KUKA KRL program: MyProgram_068().src

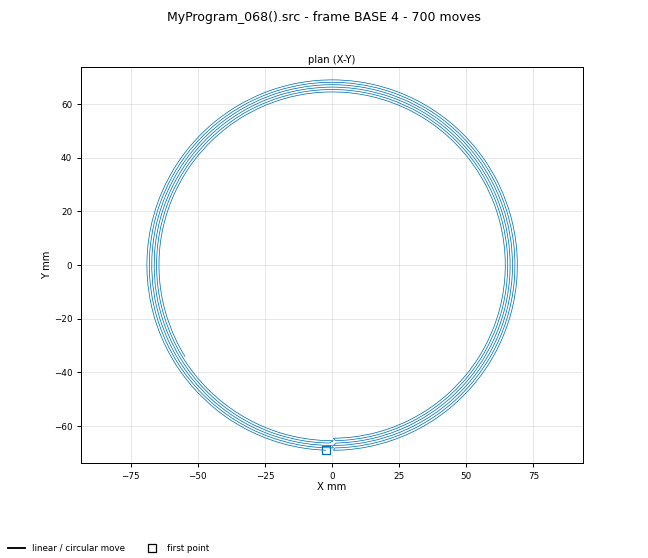
[picture p0: tool path of MyProgram_068().src in frame BASE 4, 700 of 700 moves have a stored position in this frame; points joined in program order, loops and branches not executed]
&ACCESS RVP
&REL 1
&PARAM TEMPLATE = C:\KRC\Roboter\Template\vorgabe
&PARAM EDITMASK = *
DEF MyProgram_068()
; ---- Setting reference (Base) ----
$BASE = BASE_DATA[4]

; --------------------------
; ---- Setting tool (TCP) ----
$TOOL = TOOL_DATA[3]
; --------------------------

$VEL.CP = VEL_APROX_PRINT
Startdeposition()
$VEL.CP = VEL_PRINT
LIN {X -2.4169,Y -68.9685,Z 75,A -97.7001,B 24.906,C -2.2384,E1 24.9936,E2 -177.965} C_DIS
LIN {X -6.7718,Y -68.6771,Z 75,A -101.3764,B 24.9061,C -2.2371,E1 24.9834,E2 -174.2842} C_DIS
LIN {X -9.1788,Y -68.3972,Z 75,A -103.4041,B 24.9061,C -2.2371,E1 24.9777,E2 -172.2549} C_DIS
LIN {X -12.2658,Y -67.9113,Z 75,A -106.3627,B 24.9068,C -2.2291,E1 24.9695,E2 -169.2747} C_DIS
LIN {X -15.7855,Y -67.181,Z 75,A -108.8346,B 24.9057,C -2.2426,E1 24.9629,E2 -166.8319} C_DIS
LIN {X -17.9152,Y -66.6442,Z 75,A -111.3209,B 24.9069,C -2.2281,E1 24.9561,E2 -164.3072} C_DIS
LIN {X -20.9966,Y -65.7389,Z 75,A -114.0064,B 24.9067,C -2.2296,E1 24.9489,E2 -161.6206} C_DIS
LIN {X -24.5799,Y -64.4845,Z 75,A -116.6949,B 24.9056,C -2.2431,E1 24.9419,E2 -158.9589} C_DIS
LIN {X -28.1955,Y -62.9876,Z 75,A -120.4389,B 24.9063,C -2.2351,E1 24.9322,E2 -155.187} C_DIS
LIN {X -31.9464,Y -61.1709,Z 75,A -123.1207,B 24.9044,C -2.2571,E1 24.9257,E2 -152.5506} C_DIS
LIN {X -33.7019,Y -60.2211,Z 75,A -125.4044,B 24.9055,C -2.245,E1 24.92,E2 -150.2315} C_DIS
LIN {X -37.4481,Y -57.9661,Z 75,A -128.5714,B 24.9041,C -2.2608,E1 24.9125,E2 -147.0923} C_DIS
LIN {X -39.6579,Y -56.4778,Z 75,A -131.4501,B 24.9051,C -2.2494,E1 24.9058,E2 -144.1767} C_DIS
LIN {X -42.7083,Y -54.2071,Z 75,A -134.5296,B 24.9045,C -2.2567,E1 24.899,E2 -141.1033} C_DIS
LIN {X -45.1659,Y -52.1779,Z 75,A -137.5073,B 24.9047,C -2.2544,E1 24.8927,E2 -138.1086} C_DIS
LIN {X -50.0115,Y -47.5541,Z 75,A -142.1725,B 24.902,C -2.2855,E1 24.8835,E2 -133.498} C_DIS
LIN {X -52.2098,Y -45.1287,Z 75,A -144.8753,B 24.9015,C -2.2919,E1 24.8785,E2 -130.7982} C_DIS
LIN {X -54.874,Y -41.8492,Z 75,A -148.4506,B 24.9009,C -2.2985,E1 24.8722,E2 -127.2221} C_DIS
LIN {X -56.1233,Y -40.157,Z 75,A -150.636,B 24.9013,C -2.2933,E1 24.8686,E2 -125.0136} C_DIS
LIN {X -57.9622,Y -37.4542,Z 75,A -153.0207,B 24.9001,C -2.3072,E1 24.8649,E2 -122.6502} C_DIS
LIN {X -59.1194,Y -35.6002,Z 75,A -156.0291,B 24.9019,C -2.2866,E1 24.8605,E2 -119.5771} C_DIS
LIN {X -61.0804,Y -32.1183,Z 75,A -159.2393,B 24.9009,C -2.2978,E1 24.8563,E2 -116.3766} C_DIS
LIN {X -62.7279,Y -28.7708,Z 75,A -161.5557,B 24.8988,C -2.3228,E1 24.8537,E2 -114.1072} C_DIS
LIN {X -64.116,Y -25.5271,Z 75,A -165.1655,B 24.8993,C -2.3169,E1 24.8498,E2 -110.4633} C_DIS
LIN {X -65.2783,Y -22.3892,Z 75,A -167.2138,B 24.8972,C -2.3402,E1 24.848,E2 -108.459} C_DIS
LIN {X -66.2797,Y -19.22,Z 75,A -169.9974,B 24.8966,C -2.3479,E1 24.8457,E2 -105.6777} C_DIS
LIN {X -67.1155,Y -16.059,Z 75,A -173.0277,B 24.8964,C -2.3495,E1 24.8436,E2 -102.6337} C_DIS
LIN {X -67.8136,Y -12.7977,Z 75,A -176.0352,B 24.8961,C -2.3531,E1 24.842,E2 -99.6169} C_DIS
LIN {X -68.5949,Y -7.5688,Z 75,A 178.9947,B 24.8959,C -2.3549,E1 24.8403,E2 -94.6213} C_DIS
LIN {X -68.9256,Y -3.4354,Z 75,A 176.9644,B 24.8924,C -2.3948,E1 24.84,E2 -92.6742} C_DIS
LIN {X -69.0119,Y -0.1041,Z 75,A 173.4964,B 24.8929,C -2.389,E1 24.8398,E2 -89.1714} C_DIS
LIN {X -68.9341,Y 3.2516,Z 75,A 170.7988,B 24.8919,C -2.3997,E1 24.8401,E2 -86.4831} C_DIS
LIN {X -68.597,Y 7.5488,Z 75,A 167.4395,B 24.8905,C -2.4155,E1 24.8409,E2 -83.1416} C_DIS
LIN {X -67.9375,Y 12.1205,Z 75,A 163.8781,B 24.8889,C -2.4334,E1 24.8424,E2 -79.6015} C_DIS
LIN {X -67.0696,Y 16.2506,Z 75,A 160.4913,B 24.8876,C -2.4468,E1 24.8444,E2 -76.2268} C_DIS
LIN {X -65.8431,Y 20.6675,Z 75,A 155.409,B 24.889,C -2.4322,E1 24.8484,E2 -71.0802} C_DIS
LIN {X -64.756,Y 23.8555,Z 75,A 153.2009,B 24.8871,C -2.4528,E1 24.8504,E2 -68.9088} C_DIS
LIN {X -63.907,Y 26.044,Z 75,A 150.9864,B 24.8871,C -2.4531,E1 24.8528,E2 -66.6829} C_DIS
LIN {X -62.007,Y 30.2934,Z 75,A 147.2256,B 24.8858,C -2.4667,E1 24.8572,E2 -62.934} C_DIS
LIN {X -59.24,Y 35.3996,Z 75,A 142.4927,B 24.8843,C -2.4823,E1 24.8636,E2 -58.2136} C_DIS
LIN {X -57.2828,Y 38.4856,Z 75,A 139.4955,B 24.8835,C -2.4915,E1 24.8682,E2 -55.2232} C_DIS
LIN {X -55.3718,Y 41.1877,Z 75,A 136.6952,B 24.8829,C -2.4977,E1 24.8728,E2 -52.4242} C_DIS
LIN {X -52.9777,Y 44.2243,Z 75,A 133.2143,B 24.8827,C -2.5003,E1 24.8789,E2 -48.9333} C_DIS
LIN {X -49.893,Y 47.6778,Z 75,A 130.0717,B 24.8803,C -2.5248,E1 24.8848,E2 -45.8351} C_DIS
LIN {X -47.8354,Y 49.7411,Z 75,A 126.9391,B 24.8812,C -2.5152,E1 24.8911,E2 -42.6666} C_DIS
LIN {X -45.1609,Y 52.1823,Z 75,A 123.1647,B 24.8822,C -2.5056,E1 24.8991,E2 -38.8544} C_DIS
LIN {X -41.8434,Y 54.8786,Z 75,A 119.5436,B 24.8816,C -2.5114,E1 24.9072,E2 -35.2341} C_DIS
LIN {X -38.259,Y 57.4348,Z 75,A 117.3549,B 24.8779,C -2.5502,E1 24.912,E2 -33.1306} C_DIS
LIN {X -35.8964,Y 58.9394,Z 75,A 114.595,B 24.8784,C -2.545,E1 24.9186,E2 -30.3494} C_DIS
LIN {X -32.8881,Y 60.6694,Z 75,A 111.7508,B 24.8779,C -2.5507,E1 24.9255,E2 -27.5107} C_DIS
LIN {X -27.9982,Y 63.0765,Z 75,A 106.5089,B 24.8787,C -2.5418,E1 24.9388,E2 -22.2343} C_DIS
LIN {X -24.9034,Y 64.3605,Z 75,A 104.6486,B 24.8764,C -2.5661,E1 24.9435,E2 -20.4278} C_DIS
LIN {X -22.9342,Y 65.0879,Z 75,A 102.0329,B 24.8781,C -2.5487,E1 24.9505,E2 -17.7655} C_DIS
LIN {X -19.8759,Y 66.0858,Z 75,A 99.9814,B 24.8764,C -2.5656,E1 24.9559,E2 -15.7507} C_DIS
LIN {X -15.4692,Y 67.254,Z 75,A 96.1652,B 24.8761,C -2.5685,E1 24.9662,E2 -11.9361} C_DIS
LIN {X -13.1799,Y 67.74,Z 75,A 93.4317,B 24.8777,C -2.552,E1 24.9739,E2 -9.1603} C_DIS
LIN {X -9.5408,Y 68.3476,Z 75,A 91.278,B 24.8755,C -2.5749,E1 24.9797,E2 -7.0592} C_DIS
LIN {X -6.6273,Y 68.6918,Z 75,A 88.761,B 24.8755,C -2.5743,E1 24.9866,E2 -4.5394} C_DIS
LIN {X -4.354,Y 68.8733,Z 75,A 85.9582,B 24.8776,C -2.5539,E1 24.9946,E2 -1.6871} C_DIS
LIN {X -0.5063,Y 69.0083,Z 75,A 83.6802,B 24.8754,C -2.5762,E1 25.0008,E2 0.5381} C_DIS
LIN {X 2.5422,Y 68.9643,Z 75,A 81.1062,B 24.8754,C -2.5754,E1 25.008,E2 3.1135} C_DIS
LIN {X 7.1724,Y 68.6364,Z 75,A 76.1587,B 24.878,C -2.5492,E1 25.0219,E2 8.1203} C_DIS
LIN {X 11.5572,Y 68.0357,Z 75,A 73.6683,B 24.8754,C -2.5764,E1 25.0286,E2 10.5438} C_DIS
LIN {X 14.4514,Y 67.4806,Z 75,A 70.6369,B 24.8769,C -2.5611,E1 25.037,E2 13.6075} C_DIS
LIN {X 17.8736,Y 66.6555,Z 75,A 67.8581,B 24.8767,C -2.5628,E1 25.0445,E2 16.378} C_DIS
LIN {X 21.6874,Y 65.5149,Z 75,A 65.1206,B 24.8756,C -2.5742,E1 25.0517,E2 19.0834} C_DIS
LIN {X 25.2023,Y 64.2436,Z 75,A 61.4768,B 24.8772,C -2.558,E1 25.0613,E2 22.758} C_DIS
LIN {X 29.4402,Y 62.4163,Z 75,A 58.0247,B 24.8767,C -2.5632,E1 25.07,E2 26.1892} C_DIS
LIN {X 32.7358,Y 60.752,Z 75,A 54.8729,B 24.8773,C -2.557,E1 25.0778,E2 29.3467} C_DIS
LIN {X 36.1577,Y 58.7806,Z 75,A 51.9971,B 24.8767,C -2.5626,E1 25.0847,E2 32.2007} C_DIS
LIN {X 39.1022,Y 56.864,Z 75,A 48.3317,B 24.879,C -2.5388,E1 25.0933,E2 35.9101} C_DIS
LIN {X 42.6741,Y 54.2341,Z 75,A 44.6835,B 24.8795,C -2.5332,E1 25.1014,E2 39.5582} C_DIS
LIN {X 45.0638,Y 52.2668,Z 75,A 42.5551,B 24.8789,C -2.5397,E1 25.1059,E2 41.6631} C_DIS
LIN {X 47.8326,Y 49.7438,Z 75,A 40.0156,B 24.8781,C -2.5484,E1 25.111,E2 44.1717} C_DIS
LIN {X 49.9659,Y 47.6021,Z 75,A 36.8259,B 24.8803,C -2.5252,E1 25.1173,E2 47.4026} C_DIS
LIN {X 53.072,Y 44.1108,Z 75,A 33.3588,B 24.8801,C -2.5273,E1 25.1237,E2 50.8491} C_DIS
LIN {X 55.6965,Y 40.7468,Z 75,A 28.9517,B 24.8831,C -2.496,E1 25.1312,E2 55.3092} C_DIS
LIN {X 57.6972,Y 37.861,Z 75,A 26.2056,B 24.8833,C -2.4931,E1 25.1354,E2 58.0486} C_DIS
LIN {X 60.3606,Y 33.4522,Z 75,A 22.0953,B 24.884,C -2.4862,E1 25.1411,E2 62.154} C_DIS
LIN {X 61.8517,Y 30.6067,Z 75,A 19.7892,B 24.8838,C -2.4886,E1 25.144,E2 64.4421} C_DIS
LIN {X 63.6158,Y 26.7475,Z 75,A 15.7389,B 24.886,C -2.4645,E1 25.1486,E2 68.5272} C_DIS
LIN {X 65.6592,Y 21.2431,Z 75,A 11.2518,B 24.8864,C -2.4607,E1 25.1527,E2 72.9981} C_DIS
LIN {X 66.648,Y 17.9012,Z 75,A 8.3955,B 24.8871,C -2.4531,E1 25.1549,E2 75.8561} C_DIS
LIN {X 67.5009,Y 14.3579,Z 75,A 5.5509,B 24.8875,C -2.4488,E1 25.1567,E2 78.6943} C_DIS
LIN {X 68.1413,Y 10.9181,Z 75,A 2.6382,B 24.8883,C -2.4396,E1 25.1581,E2 81.6117} C_DIS
LIN {X 68.6615,Y 6.9308,Z 75,A -0.3525,B 24.8883,C -2.4387,E1 25.1591,E2 84.5868} C_DIS
LIN {X 68.8098,Y 5.2596,Z 75,A -2.8449,B 24.8915,C -2.4044,E1 25.1596,E2 87.1454} C_DIS
LIN {X 68.9925,Y 1.593,Z 75,A -4.6966,B 24.8894,C -2.4273,E1 25.1598,E2 88.932} C_DIS
LIN {X 68.9365,Y -3.1965,Z 75,A -8.6973,B 24.8906,C -2.414,E1 25.1596,E2 92.9404} C_DIS
LIN {X 68.7647,Y -5.8221,Z 75,A -11.1863,B 24.892,C -2.3987,E1 25.1591,E2 95.4508} C_DIS
LIN {X 68.4631,Y -8.6741,Z 75,A -13.9477,B 24.8936,C -2.3808,E1 25.1581,E2 98.2382} C_DIS
LIN {X 67.7432,Y -13.1634,Z 75,A -17.5482,B 24.8943,C -2.3736,E1 25.1564,E2 101.8345} C_DIS
LIN {X 66.9693,Y -16.6615,Z 75,A -21.103,B 24.8965,C -2.3485,E1 25.154,E2 105.4279} C_DIS
LIN {X 65.9661,Y -20.2695,Z 75,A -23.5037,B 24.8957,C -2.3581,E1 25.1521,E2 107.7924} C_DIS
LIN {X 64.4258,Y -24.734,Z 75,A -27.5665,B 24.8971,C -2.3423,E1 25.1482,E2 111.8698} C_DIS
LIN {X 63.1759,Y -27.7714,Z 75,A -29.6765,B 24.8963,C -2.3509,E1 25.1459,E2 113.9479} C_DIS
LIN {X 61.2105,Y -31.8713,Z 75,A -34.8597,B 24.9006,C -2.3018,E1 25.1393,E2 119.2194} C_DIS
LIN {X 58.9736,Y -35.8402,Z 75,A -37.1636,B 24.8981,C -2.3308,E1 25.1362,E2 121.443} C_DIS
LIN {X 57.6967,Y -37.8618,Z 75,A -39.7177,B 24.8999,C -2.3099,E1 25.1322,E2 124.0336} C_DIS
LIN {X 55.38,Y -41.1773,Z 75,A -43.2595,B 24.9011,C -2.2959,E1 25.1264,E2 127.5914} C_DIS
LIN {X 52.7711,Y -44.4719,Z 75,A -46.2238,B 24.9007,C -2.3009,E1 25.1212,E2 130.5303} C_DIS
LIN {X 50.6612,Y -46.8606,Z 75,A -49.3423,B 24.9023,C -2.2817,E1 25.1153,E2 133.6804} C_DIS
LIN {X 46.7275,Y -50.7833,Z 75,A -53.2212,B 24.9016,C -2.2903,E1 25.1076,E2 137.5227} C_DIS
LIN {X 44.812,Y -52.4813,Z 75,A -55.5297,B 24.9024,C -2.2806,E1 25.1027,E2 139.845} C_DIS
LIN {X 42.6119,Y -54.2833,Z 75,A -58.3498,B 24.9039,C -2.2634,E1 25.0964,E2 142.6952} C_DIS
LIN {X 39.0721,Y -56.884,Z 75,A -61.6881,B 24.9039,C -2.2642,E1 25.0889,E2 146.0202} C_DIS
LIN {X 36.8921,Y -58.3226,Z 75,A -63.7241,B 24.9039,C -2.2635,E1 25.0841,E2 148.0512} C_DIS
LIN {X 34.1032,Y -59.9956,Z 75,A -67.0204,B 24.9056,C -2.2432,E1 25.076,E2 151.3856} C_DIS
LIN {X 30.9176,Y -61.6976,Z 75,A -70.0425,B 24.9061,C -2.2377,E1 25.0685,E2 154.4125} C_DIS
LIN {X 27.9422,Y -63.1014,Z 75,A -72.1201,B 24.905,C -2.2503,E1 25.0633,E2 156.4551} C_DIS
LIN {X 24.0168,Y -64.6973,Z 75,A -76.0525,B 24.9063,C -2.2349,E1 25.053,E2 160.4153} C_DIS
LIN {X 20.2897,Y -65.9602,Z 75,A -79.1443,B 24.9063,C -2.2355,E1 25.0448,E2 163.4999} C_DIS
LIN {X 15.7939,Y -67.179,Z 75,A -82.7107,B 24.9059,C -2.2392,E1 25.0352,E2 167.0521} C_DIS
LIN {X 11.2615,Y -68.0852,Z 75,A -86.5874,B 24.9063,C -2.2351,E1 25.0245,E2 170.9341} C_DIS
LIN {X 6.7327,Y -68.682,Z 75,A -90.3445,B 24.9064,C -2.2337,E1 25.0141,E2 174.6918} C_DIS
LIN {X 3.7919,Y -68.9059,Z 75,A -92.7846,B 24.9064,C -2.2328,E1 25.0073,E2 177.1329} C_DIS
LIN {X 0.4755,Y -68.972,Z 75,A -95.369,B 24.9061,C -2.2368,E1 25.0001,E2 179.7074} C_DIS
Enddeposition()
LIN {X 0.4755,Y -68.972,Z 75,A -95.369,B 24.9061,C -2.2368,E1 25.0001,E2 179.7074} C_DIS
Startdeposition()
$VEL.CP = VEL_PRINT
LIN {X 1.0869,Y -68.1022,Z 75,A -94.0872,B 24.9033,C -2.2708,E1 25.0039,E2 178.3451} C_DIS
LIN {X 3.4577,Y -68.0236,Z 75,A -91.8539,B 24.9027,C -2.2774,E1 25.0102,E2 176.0968} C_DIS
LIN {X 6.6528,Y -67.7862,Z 75,A -88.3869,B 24.9009,C -2.2981,E1 25.02,E2 172.5825} C_DIS
LIN {X 10.0513,Y -67.3654,Z 75,A -86.5018,B 24.9029,C -2.275,E1 25.025,E2 170.7541} C_DIS
LIN {X 14.6106,Y -66.5253,Z 75,A -82.5987,B 24.9026,C -2.2782,E1 25.0357,E2 166.8478} C_DIS
LIN {X 18.2097,Y -65.6324,Z 75,A -78.8592,B 24.901,C -2.2972,E1 25.0459,E2 163.069} C_DIS
LIN {X 21.6851,Y -64.5665,Z 75,A -75.0694,B 24.899,C -2.32,E1 25.0561,E2 159.2326} C_DIS
LIN {X 25.838,Y -63.0198,Z 75,A -72.1076,B 24.9003,C -2.3051,E1 25.0637,E2 156.3128} C_DIS
LIN {X 29.4896,Y -61.3957,Z 75,A -69.1878,B 24.9009,C -2.2988,E1 25.071,E2 153.4155} C_DIS
LIN {X 31.9355,Y -60.1602,Z 75,A -66.8974,B 24.9006,C -2.3022,E1 25.0767,E2 151.1232} C_DIS
LIN {X 34.9587,Y -58.4558,Z 75,A -63.9982,B 24.9002,C -2.3069,E1 25.0837,E2 148.2217} C_DIS
LIN {X 38.1825,Y -56.4018,Z 75,A -60.5693,B 24.8991,C -2.3187,E1 25.0917,E2 144.7761} C_DIS
LIN {X 41.0965,Y -54.3157,Z 75,A -57.5071,B 24.8985,C -2.3262,E1 25.0986,E2 141.7072} C_DIS
LIN {X 43.9939,Y -51.9967,Z 75,A -54.6941,B 24.8985,C -2.3248,E1 25.1047,E2 138.9082} C_DIS
LIN {X 45.5482,Y -50.6405,Z 75,A -52.7532,B 24.8978,C -2.3342,E1 25.1087,E2 136.9526} C_DIS
LIN {X 48.0466,Y -48.2769,Z 75,A -50.0508,B 24.8976,C -2.336,E1 25.1141,E2 134.2574} C_DIS
LIN {X 50.5842,Y -45.611,Z 75,A -47.0184,B 24.8971,C -2.3419,E1 25.1199,E2 131.2242} C_DIS
LIN {X 52.5069,Y -43.3836,Z 75,A -44.2671,B 24.8959,C -2.3558,E1 25.1249,E2 128.4529} C_DIS
LIN {X 54.7777,Y -40.4791,Z 75,A -41.181,B 24.8952,C -2.3636,E1 25.1301,E2 125.3629} C_DIS
LIN {X 57.5942,Y -36.3604,Z 75,A -37.5141,B 24.8954,C -2.3607,E1 25.1358,E2 121.721} C_DIS
LIN {X 59.0494,Y -33.9447,Z 75,A -34.8729,B 24.8942,C -2.3748,E1 25.1395,E2 119.0601} C_DIS
LIN {X 60.4973,Y -31.2932,Z 75,A -32.3896,B 24.8937,C -2.3806,E1 25.1428,E2 116.5762} C_DIS
LIN {X 61.731,Y -28.7812,Z 75,A -30.1209,B 24.8932,C -2.3852,E1 25.1455,E2 114.3087} C_DIS
LIN {X 62.7941,Y -26.3812,Z 75,A -27.627,B 24.8919,C -2.3997,E1 25.1483,E2 111.7944} C_DIS
LIN {X 64.3255,Y -22.3903,Z 75,A -24.4101,B 24.8919,C -2.4002,E1 25.1514,E2 108.5941} C_DIS
LIN {X 65.4179,Y -18.9657,Z 75,A -20.7689,B 24.8895,C -2.4266,E1 25.1544,E2 104.9113} C_DIS
LIN {X 66.4072,Y -15.1392,Z 75,A -17.7154,B 24.8892,C -2.4295,E1 25.1563,E2 101.8687} C_DIS
LIN {X 67.1595,Y -11.3437,Z 75,A -14.749,B 24.889,C -2.4318,E1 25.1578,E2 98.9142} C_DIS
LIN {X 67.6452,Y -7.9495,Z 75,A -12.1774,B 24.889,C -2.4324,E1 25.1588,E2 96.3564} C_DIS
LIN {X 67.8379,Y -6.0923,Z 75,A -10.3259,B 24.8878,C -2.4451,E1 25.1593,E2 94.4859} C_DIS
LIN {X 68.0448,Y -2.9954,Z 75,A -7.9509,B 24.8876,C -2.4469,E1 25.1597,E2 92.1207} C_DIS
LIN {X 68.0927,Y 1.6027,Z 75,A -4.3439,B 24.8872,C -2.4519,E1 25.1597,E2 88.5232} C_DIS
LIN {X 67.8357,Y 6.1162,Z 75,A 0.0289,B 24.8846,C -2.4795,E1 25.1589,E2 84.1113} C_DIS
LIN {X 67.5084,Y 9.0431,Z 75,A 2.642,B 24.8835,C -2.491,E1 25.158,E2 81.4865} C_DIS
LIN {X 66.6843,Y 13.8673,Z 75,A 6.4399,B 24.8832,C -2.4949,E1 25.1561,E2 77.7017} C_DIS
LIN {X 65.3548,Y 19.1795,Z 75,A 10.8866,B 24.8823,C -2.5043,E1 25.153,E2 73.2581} C_DIS
LIN {X 63.9617,Y 23.4088,Z 75,A 14.751,B 24.8809,C -2.5185,E1 25.1495,E2 69.382} C_DIS
LIN {X 62.5623,Y 26.9281,Z 75,A 18.2459,B 24.8793,C -2.536,E1 25.1457,E2 65.8651} C_DIS
LIN {X 60.827,Y 30.648,Z 75,A 21.9802,B 24.8776,C -2.5531,E1 25.1411,E2 62.1103} C_DIS
LIN {X 58.6332,Y 34.6586,Z 75,A 25.2658,B 24.8781,C -2.5482,E1 25.1366,E2 58.8533} C_DIS
LIN {X 56.754,Y 37.6576,Z 75,A 27.8055,B 24.8785,C -2.5441,E1 25.1328,E2 56.3361} C_DIS
LIN {X 54.7612,Y 40.5017,Z 75,A 31.5931,B 24.8756,C -2.5744,E1 25.1265,E2 52.4952} C_DIS
LIN {X 52.4107,Y 43.4993,Z 75,A 34.9365,B 24.8745,C -2.5855,E1 25.1206,E2 49.1409} C_DIS
LIN {X 50.2652,Y 45.9618,Z 75,A 36.5896,B 24.8767,C -2.5626,E1 25.1176,E2 47.5493} C_DIS
LIN {X 47.4872,Y 48.8275,Z 75,A 39.9639,B 24.876,C -2.5701,E1 25.111,E2 44.1717} C_DIS
LIN {X 44.8543,Y 51.2559,Z 75,A 42.7745,B 24.876,C -2.5709,E1 25.1053,E2 41.3706} C_DIS
LIN {X 42,Y 53.6205,Z 75,A 46.0803,B 24.8749,C -2.5815,E1 25.0981,E2 38.0523} C_DIS
LIN {X 39.2161,Y 55.6896,Z 75,A 50.0343,B 24.8718,C -2.6132,E1 25.089,E2 34.0371} C_DIS
LIN {X 36.5015,Y 57.505,Z 75,A 52.0993,B 24.8731,C -2.5999,E1 25.0843,E2 32.0104} C_DIS
LIN {X 34.0059,Y 59.0141,Z 75,A 54.7274,B 24.8723,C -2.6078,E1 25.0779,E2 29.3714} C_DIS
LIN {X 29.7678,Y 61.262,Z 75,A 58.4606,B 24.8726,C -2.6053,E1 25.0687,E2 25.6546} C_DIS
LIN {X 27.3322,Y 62.3862,Z 75,A 60.9801,B 24.8717,C -2.6144,E1 25.0622,E2 23.1197} C_DIS
LIN {X 23.6527,Y 63.8718,Z 75,A 64.3404,B 24.8713,C -2.6182,E1 25.0534,E2 19.7579} C_DIS
LIN {X 20.4574,Y 64.9666,Z 75,A 67.5673,B 24.8701,C -2.63,E1 25.0448,E2 16.5088} C_DIS
LIN {X 17.1421,Y 65.9186,Z 75,A 70.4294,B 24.8701,C -2.6308,E1 25.0371,E2 13.6493} C_DIS
LIN {X 12.4844,Y 66.958,Z 75,A 74.3353,B 24.8701,C -2.6298,E1 25.0264,E2 9.7504} C_DIS
LIN {X 6.9767,Y 67.7526,Z 75,A 78.7301,B 24.8707,C -2.6238,E1 25.0143,E2 5.3735} C_DIS
LIN {X 3.13,Y 68.0391,Z 75,A 81.7715,B 24.8712,C -2.6189,E1 25.0058,E2 2.3449} C_DIS
LIN {X -0.0016,Y 68.1119,Z 75,A 85.1275,B 24.8696,C -2.6357,E1 24.9964,E2 -1.0508} C_DIS
LIN {X -4.7805,Y 67.943,Z 75,A 88.9222,B 24.8702,C -2.6287,E1 24.9858,E2 -4.83} C_DIS
LIN {X -9.1383,Y 67.496,Z 75,A 93.0135,B 24.8695,C -2.6362,E1 24.9744,E2 -8.9419} C_DIS
LIN {X -12.7415,Y 66.9085,Z 75,A 95.0491,B 24.8721,C -2.6096,E1 24.969,E2 -10.9165} C_DIS
LIN {X -17.915,Y 65.7126,Z 75,A 99.6489,B 24.8722,C -2.6085,E1 24.9565,E2 -15.5199} C_DIS
LIN {X -21.2781,Y 64.7025,Z 75,A 102.4982,B 24.8728,C -2.6028,E1 24.949,E2 -18.3605} C_DIS
LIN {X -25.0973,Y 63.3185,Z 75,A 106.4735,B 24.872,C -2.611,E1 24.9385,E2 -22.3637} C_DIS
LIN {X -29.5209,Y 61.3807,Z 75,A 110.5312,B 24.8726,C -2.6048,E1 24.9282,E2 -26.4167} C_DIS
LIN {X -32.2641,Y 59.9846,Z 75,A 112.7631,B 24.8738,C -2.5925,E1 24.9228,E2 -28.6255} C_DIS
LIN {X -36.9014,Y 57.2484,Z 75,A 116.8402,B 24.8756,C -2.5744,E1 24.9131,E2 -32.6718} C_DIS
LIN {X -38.4899,Y 56.1932,Z 75,A 119.028,B 24.8746,C -2.5841,E1 24.9079,E2 -34.89} C_DIS
LIN {X -41.1422,Y 54.2815,Z 75,A 121.9427,B 24.8748,C -2.582,E1 24.9014,E2 -37.8103} C_DIS
LIN {X -44.6967,Y 51.3936,Z 75,A 125.4343,B 24.8764,C -2.5658,E1 24.894,E2 -41.2765} C_DIS
LIN {X -47.477,Y 48.8357,Z 75,A 128.981,B 24.8764,C -2.5664,E1 24.8867,E2 -44.8392} C_DIS
LIN {X -50.34,Y 45.8803,Z 75,A 132.5946,B 24.8768,C -2.5612,E1 24.8798,E2 -48.4562} C_DIS
LIN {X -52.6576,Y 43.202,Z 75,A 135.0195,B 24.8787,C -2.5417,E1 24.8755,E2 -50.8457} C_DIS
LIN {X -54.5114,Y 40.836,Z 75,A 137.9229,B 24.8786,C -2.5431,E1 24.8706,E2 -53.7661} C_DIS
LIN {X -56.3584,Y 38.2466,Z 75,A 140.3689,B 24.8798,C -2.531,E1 24.8667,E2 -56.1952} C_DIS
LIN {X -58.5741,Y 34.7586,Z 75,A 144.3742,B 24.8796,C -2.5324,E1 24.8608,E2 -60.2245} C_DIS
LIN {X -60.9103,Y 30.4806,Z 75,A 148.0247,B 24.8816,C -2.5111,E1 24.8561,E2 -63.8434} C_DIS
LIN {X -63.2214,Y 25.3427,Z 75,A 152.859,B 24.8828,C -2.4989,E1 24.8507,E2 -68.6753} C_DIS
LIN {X -64.4088,Y 22.1528,Z 75,A 155.8482,B 24.8834,C -2.4928,E1 24.8479,E2 -71.6668} C_DIS
LIN {X -65.1652,Y 19.8148,Z 75,A 158.6799,B 24.8824,C -2.5025,E1 24.8455,E2 -74.5381} C_DIS
LIN {X -66.1246,Y 16.3294,Z 75,A 160.4448,B 24.8858,C -2.4663,E1 24.8444,E2 -76.2268} C_DIS
LIN {X -66.8466,Y 13.063,Z 75,A 163.6249,B 24.886,C -2.4651,E1 24.8425,E2 -79.4225} C_DIS
LIN {X -67.593,Y 8.3896,Z 75,A 167.6803,B 24.887,C -2.454,E1 24.8408,E2 -83.4757} C_DIS
LIN {X -67.9481,Y 4.7042,Z 75,A 170.8745,B 24.8877,C -2.4458,E1 24.8401,E2 -86.6694} C_DIS
LIN {X -68.1071,Y -0.8122,Z 75,A 175.6239,B 24.8889,C -2.4333,E1 24.8398,E2 -91.4175} C_DIS
LIN {X -67.9649,Y -4.456,Z 75,A 178.8493,B 24.8895,C -2.4269,E1 24.8403,E2 -94.6471} C_DIS
LIN {X -67.6974,Y -7.5037,Z 75,A -178.4767,B 24.89,C -2.421,E1 24.8411,E2 -97.3229} C_DIS
LIN {X -67.0393,Y -12.0335,Z 75,A -174.8549,B 24.8915,C -2.4043,E1 24.8427,E2 -100.9263} C_DIS
LIN {X -66.5908,Y -14.31,Z 75,A -172.1847,B 24.8907,C -2.4135,E1 24.8443,E2 -103.6345} C_DIS
LIN {X -65.8087,Y -17.5594,Z 75,A -169.5071,B 24.8917,C -2.4022,E1 24.8462,E2 -106.3006} C_DIS
LIN {X -64.6834,Y -21.3372,Z 75,A -166.9833,B 24.8941,C -2.3756,E1 24.8482,E2 -108.7753} C_DIS
LIN {X -63.597,Y -24.3837,Z 75,A -163.657,B 24.8937,C -2.3806,E1 24.8515,E2 -112.1322} C_DIS
LIN {X -62.0914,Y -27.9951,Z 75,A -160.6172,B 24.895,C -2.3659,E1 24.8549,E2 -115.1539} C_DIS
LIN {X -60.7282,Y -30.8413,Z 75,A -158.1192,B 24.8959,C -2.3553,E1 24.8579,E2 -117.64} C_DIS
LIN {X -58.4274,Y -35.0068,Z 75,A -153.9782,B 24.8966,C -2.3476,E1 24.8637,E2 -121.7842} C_DIS
LIN {X -56.5051,Y -38.0299,Z 75,A -150.6916,B 24.8967,C -2.3459,E1 24.8687,E2 -125.0834} C_DIS
LIN {X -54.2437,Y -41.1924,Z 75,A -147.186,B 24.897,C -2.3432,E1 24.8746,E2 -128.5993} C_DIS
LIN {X -51.4938,Y -44.5818,Z 75,A -143.5295,B 24.8977,C -2.3345,E1 24.8811,E2 -132.2518} C_DIS
LIN {X -49.3518,Y -46.9427,Z 75,A -140.6013,B 24.8977,C -2.3342,E1 24.8868,E2 -135.1921} C_DIS
LIN {X -47.0833,Y -49.2168,Z 75,A -138.7691,B 24.8999,C -2.3093,E1 24.8904,E2 -136.9725} C_DIS
LIN {X -44.3466,Y -51.6962,Z 75,A -135.8753,B 24.9009,C -2.2985,E1 24.8963,E2 -139.8522} C_DIS
LIN {X -41.6336,Y -53.9047,Z 75,A -132.853,B 24.9012,C -2.2949,E1 24.9029,E2 -142.8773} C_DIS
LIN {X -39.9883,Y -55.1371,Z 75,A -130.3372,B 24.8999,C -2.3098,E1 24.9087,E2 -145.4373} C_DIS
LIN {X -36.9713,Y -57.2035,Z 75,A -127.5312,B 24.9009,C -2.2988,E1 24.9152,E2 -148.2263} C_DIS
LIN {X -34.8367,Y -58.5279,Z 75,A -125.1198,B 24.9005,C -2.3026,E1 24.921,E2 -150.6542} C_DIS
LIN {X -31.3204,Y -60.4833,Z 75,A -122.2449,B 24.9019,C -2.2865,E1 24.928,E2 -153.4986} C_DIS
LIN {X -28.526,Y -61.8498,Z 75,A -119.3888,B 24.9017,C -2.289,E1 24.9352,E2 -156.3681} C_DIS
LIN {X -24.7168,Y -63.468,Z 75,A -116.0656,B 24.9023,C -2.2818,E1 24.9438,E2 -159.6817} C_DIS
LIN {X -20.5191,Y -64.9473,Z 75,A -112.2598,B 24.9024,C -2.2803,E1 24.9539,E2 -163.491} C_DIS
LIN {X -16.3678,Y -66.1152,Z 75,A -108.7645,B 24.9029,C -2.2749,E1 24.9633,E2 -166.9788} C_DIS
LIN {X -12.4758,Y -66.9584,Z 75,A -104.9728,B 24.9021,C -2.2842,E1 24.9737,E2 -170.7969} C_DIS
LIN {X -8.9685,Y -67.5175,Z 75,A -102.4061,B 24.903,C -2.2733,E1 24.9808,E2 -173.3399} C_DIS
LIN {X -7.0353,Y -67.7464,Z 75,A -99.863,B 24.9012,C -2.2953,E1 24.988,E2 -175.9366} C_DIS
LIN {X -3.4451,Y -68.0243,Z 75,A -97.9252,B 24.9034,C -2.2686,E1 24.9932,E2 -177.8116} C_DIS
LIN {X 0.4854,Y -68.0955,Z 75,A -95.9466,B 24.9061,C -2.2372,E1 24.9986,E2 -179.716} C_DIS
Enddeposition()
LIN {X 0.4854,Y -68.0955,Z 75,A -95.9466,B 24.9061,C -2.2372,E1 24.9986,E2 -179.716} C_DIS
Startdeposition()
$VEL.CP = VEL_PRINT
LIN {X -0.0032,Y -67.2115,Z 75,A -96.5518,B 24.9052,C -2.2483,E1 24.9969,E2 -179.1371} C_DIS
LIN {X -3.4713,Y -67.122,Z 75,A -99.4646,B 24.9052,C -2.2491,E1 24.9888,E2 -176.2255} C_DIS
LIN {X -8.3352,Y -66.693,Z 75,A -103.1465,B 24.9041,C -2.2607,E1 24.9786,E2 -172.569} C_DIS
LIN {X -12.1208,Y -66.1097,Z 75,A -106.7591,B 24.9047,C -2.2537,E1 24.9686,E2 -168.9363} C_DIS
LIN {X -15.6243,Y -65.3708,Z 75,A -110.4984,B 24.9059,C -2.2396,E1 24.9584,E2 -165.1585} C_DIS
LIN {X -19.5827,Y -64.2958,Z 75,A -112.8858,B 24.9036,C -2.267,E1 24.9521,E2 -162.8324} C_DIS
LIN {X -22.1344,Y -63.4621,Z 75,A -115.0832,B 24.9032,C -2.2709,E1 24.9463,E2 -160.6401} C_DIS
LIN {X -24.5949,Y -62.5496,Z 75,A -117.7121,B 24.9038,C -2.2642,E1 24.9394,E2 -157.9895} C_DIS
LIN {X -28.0216,Y -61.0918,Z 75,A -120.9726,B 24.9037,C -2.2657,E1 24.9311,E2 -154.7248} C_DIS
LIN {X -31.2364,Y -59.5118,Z 75,A -124.0226,B 24.9034,C -2.2696,E1 24.9235,E2 -151.6758} C_DIS
LIN {X -34.055,Y -57.9452,Z 75,A -126.746,B 24.903,C -2.2739,E1 24.9169,E2 -148.9547} C_DIS
LIN {X -37.3624,Y -55.8709,Z 75,A -130.7779,B 24.9038,C -2.2639,E1 24.9074,E2 -144.8857} C_DIS
LIN {X -40.4753,Y -53.6574,Z 75,A -133.9343,B 24.9032,C -2.2717,E1 24.9004,E2 -141.7365} C_DIS
LIN {X -43.2989,Y -51.4072,Z 75,A -135.8823,B 24.9006,C -2.3015,E1 24.8964,E2 -139.8522} C_DIS
LIN {X -45.1522,Y -49.7867,Z 75,A -138.4066,B 24.9011,C -2.2964,E1 24.891,E2 -137.3057} C_DIS
LIN {X -46.8449,Y -48.1974,Z 75,A -140.8461,B 24.9016,C -2.2907,E1 24.8861,E2 -134.8425} C_DIS
LIN {X -50.4736,Y -44.3827,Z 75,A -144.7135,B 24.8996,C -2.3136,E1 24.8788,E2 -131.0126} C_DIS
LIN {X -52.4134,Y -42.0741,Z 75,A -147.5571,B 24.8996,C -2.3138,E1 24.8738,E2 -128.1562} C_DIS
LIN {X -54.1989,Y -39.7471,Z 75,A -150.0906,B 24.8991,C -2.3191,E1 24.8696,E2 -125.6234} C_DIS
LIN {X -55.7238,Y -37.5796,Z 75,A -152.1225,B 24.8982,C -2.3294,E1 24.8664,E2 -123.606} C_DIS
LIN {X -56.9137,Y -35.7522,Z 75,A -154.0513,B 24.8979,C -2.3327,E1 24.8635,E2 -121.6753} C_DIS
LIN {X -58.6187,Y -32.882,Z 75,A -156.7267,B 24.8969,C -2.3437,E1 24.8597,E2 -119.0123} C_DIS
LIN {X -60.1552,Y -29.9785,Z 75,A -160.1627,B 24.8974,C -2.3383,E1 24.8553,E2 -115.545} C_DIS
LIN {X -61.4431,Y -27.2445,Z 75,A -162.9751,B 24.8972,C -2.3407,E1 24.8521,E2 -112.7228} C_DIS
LIN {X -63.5049,Y -22.0124,Z 75,A -166.9972,B 24.8946,C -2.3702,E1 24.8482,E2 -108.7486} C_DIS
LIN {X -64.2936,Y -19.5908,Z 75,A -169.6735,B 24.8949,C -2.3664,E1 24.846,E2 -106.0478} C_DIS
LIN {X -65.5795,Y -14.7255,Z 75,A -173.3541,B 24.8927,C -2.3917,E1 24.8435,E2 -102.406} C_DIS
LIN {X -66.0071,Y -12.6659,Z 75,A -175.4732,B 24.8927,C -2.3906,E1 24.8423,E2 -100.2717} C_DIS
LIN {X -66.8066,Y -7.3743,Z 75,A 179.2853,B 24.8927,C -2.3912,E1 24.8404,E2 -95.0005} C_DIS
LIN {X -67.1946,Y -1.5269,Z 75,A 174.4704,B 24.891,C -2.4106,E1 24.8398,E2 -90.2028} C_DIS
LIN {X -67.1431,Y 3.0309,Z 75,A 171.04,B 24.889,C -2.4319,E1 24.84,E2 -86.8028} C_DIS
LIN {X -66.9091,Y 6.3687,Z 75,A 168.125,B 24.8883,C -2.4397,E1 24.8407,E2 -83.889} C_DIS
LIN {X -66.5457,Y 9.4356,Z 75,A 165.2652,B 24.8879,C -2.4435,E1 24.8417,E2 -81.0212} C_DIS
LIN {X -65.8736,Y 13.344,Z 75,A 161.7364,B 24.8872,C -2.4512,E1 24.8436,E2 -77.4899} C_DIS
LIN {X -65.2471,Y 16.1313,Z 75,A 159.0478,B 24.887,C -2.4538,E1 24.8454,E2 -74.7916} C_DIS
LIN {X -64.0649,Y 20.3272,Z 75,A 155.0706,B 24.8864,C -2.4601,E1 24.8486,E2 -70.8067} C_DIS
LIN {X -62.9263,Y 23.6153,Z 75,A 153.2891,B 24.8834,C -2.4928,E1 24.8503,E2 -69.0932} C_DIS
LIN {X -61.9661,Y 26.0291,Z 75,A 150.531,B 24.8838,C -2.4885,E1 24.8532,E2 -66.3095} C_DIS
LIN {X -60.4167,Y 29.4498,Z 75,A 147.4946,B 24.8826,C -2.5012,E1 24.8568,E2 -63.2869} C_DIS
LIN {X -57.854,Y 34.2092,Z 75,A 141.9165,B 24.8832,C -2.495,E1 24.8645,E2 -57.6646} C_DIS
LIN {X -55.8659,Y 37.3697,Z 75,A 139.5756,B 24.8807,C -2.5207,E1 24.868,E2 -55.3734} C_DIS
LIN {X -53.4609,Y 40.7349,Z 75,A 135.738,B 24.8804,C -2.5237,E1 24.8743,E2 -51.5246} C_DIS
LIN {X -50.5225,Y 44.3267,Z 75,A 132.0082,B 24.879,C -2.5384,E1 24.881,E2 -47.8127} C_DIS
LIN {X -48.3217,Y 46.716,Z 75,A 129.2516,B 24.8784,C -2.5455,E1 24.8863,E2 -45.0609} C_DIS
LIN {X -45.8552,Y 49.1394,Z 75,A 126.6259,B 24.8771,C -2.559,E1 24.8915,E2 -42.4567} C_DIS
LIN {X -44.6681,Y 50.2212,Z 75,A 124.664,B 24.878,C -2.5498,E1 24.8957,E2 -40.4648} C_DIS
LIN {X -41.7644,Y 52.6603,Z 75,A 121.6852,B 24.8768,C -2.562,E1 24.9021,E2 -37.504} C_DIS
LIN {X -39.6499,Y 54.2701,Z 75,A 119.5823,B 24.876,C -2.5701,E1 24.9067,E2 -35.4129} C_DIS
LIN {X -36.8859,Y 56.1854,Z 75,A 116.8784,B 24.8751,C -2.5791,E1 24.913,E2 -32.7214} C_DIS
LIN {X -34.131,Y 57.9002,Z 75,A 113.3697,B 24.8762,C -2.5684,E1 24.9214,E2 -29.1762} C_DIS
LIN {X -30.9992,Y 59.6364,Z 75,A 110.392,B 24.8755,C -2.575,E1 24.9287,E2 -26.206} C_DIS
LIN {X -26.7498,Y 61.6589,Z 75,A 106.6456,B 24.8744,C -2.5867,E1 24.9382,E2 -22.4783} C_DIS
LIN {X -22.7594,Y 63.2412,Z 75,A 103.2767,B 24.8733,C -2.5979,E1 24.9469,E2 -19.1289} C_DIS
LIN {X -19.6684,Y 64.2695,Z 75,A 100.5329,B 24.8729,C -2.6018,E1 24.9542,E2 -16.3895} C_DIS
LIN {X -17.6822,Y 64.8438,Z 75,A 97.6542,B 24.8751,C -2.5791,E1 24.9621,E2 -13.4523} C_DIS
LIN {X -14.302,Y 65.672,Z 75,A 95.692,B 24.8727,C -2.6039,E1 24.9673,E2 -11.5466} C_DIS
LIN {X -9.6439,Y 66.5161,Z 75,A 91.8326,B 24.872,C -2.6109,E1 24.9779,E2 -7.6998} C_DIS
LIN {X -6.3945,Y 66.9067,Z 75,A 88.4896,B 24.8731,C -2.5999,E1 24.9872,E2 -4.3286} C_DIS
LIN {X -3.3375,Y 67.1292,Z 75,A 86.0752,B 24.8726,C -2.6054,E1 24.9939,E2 -1.9265} C_DIS
LIN {X 0.0082,Y 67.2125,Z 75,A 83.4593,B 24.872,C -2.6115,E1 25.0012,E2 0.675} C_DIS
LIN {X 2.3819,Y 67.1698,Z 75,A 80.3726,B 24.8743,C -2.5873,E1 25.01,E2 3.8185} C_DIS
LIN {X 5.8003,Y 66.961,Z 75,A 78.4371,B 24.8721,C -2.6099,E1 25.0152,E2 5.6994} C_DIS
LIN {X 10.0319,Y 66.4579,Z 75,A 74.6114,B 24.8726,C -2.6046,E1 25.0258,E2 9.5346} C_DIS
LIN {X 12.6969,Y 66.0011,Z 75,A 71.3363,B 24.8749,C -2.581,E1 25.035,E2 12.8619} C_DIS
LIN {X 16.5063,Y 65.1533,Z 75,A 69.0445,B 24.8727,C -2.6035,E1 25.041,E2 15.097} C_DIS
LIN {X 19.2061,Y 64.4088,Z 75,A 66.8031,B 24.8726,C -2.6054,E1 25.047,E2 17.3302} C_DIS
LIN {X 21.7408,Y 63.5985,Z 75,A 63.6457,B 24.8748,C -2.5822,E1 25.0555,E2 20.5363} C_DIS
LIN {X 27.1425,Y 61.4877,Z 75,A 59.6506,B 24.8731,C -2.6001,E1 25.0657,E2 24.4799} C_DIS
LIN {X 28.7407,Y 60.7577,Z 75,A 57.2087,B 24.8755,C -2.5754,E1 25.072,E2 26.9741} C_DIS
LIN {X 33.5025,Y 58.2661,Z 75,A 53.6124,B 24.8737,C -2.5934,E1 25.0807,E2 30.5173} C_DIS
LIN {X 35.5495,Y 57.0403,Z 75,A 51.29,B 24.8747,C -2.5833,E1 25.0862,E2 32.8565} C_DIS
LIN {X 39.0616,Y 54.695,Z 75,A 47.3197,B 24.8762,C -2.5682,E1 25.0954,E2 36.8489} C_DIS
LIN {X 41.3256,Y 53.0066,Z 75,A 44.632,B 24.8773,C -2.5569,E1 25.1014,E2 39.5535} C_DIS
LIN {X 44.1631,Y 50.6654,Z 75,A 41.6031,B 24.8776,C -2.5536,E1 25.1078,E2 42.5784} C_DIS
LIN {X 46.8468,Y 48.1956,Z 75,A 38.3616,B 24.8785,C -2.5438,E1 25.1143,E2 45.8295} C_DIS
LIN {X 49.1886,Y 45.8034,Z 75,A 36.5659,B 24.8765,C -2.5645,E1 25.1177,E2 47.5684} C_DIS
LIN {X 51.7494,Y 42.8878,Z 75,A 33.4416,B 24.8768,C -2.5618,E1 25.1234,E2 50.6851} C_DIS
LIN {X 53.2462,Y 41.0146,Z 75,A 30.2904,B 24.88,C -2.5285,E1 25.1289,E2 53.9002} C_DIS
LIN {X 55.4098,Y 38.0428,Z 75,A 27.7891,B 24.8792,C -2.5369,E1 25.1329,E2 56.3693} C_DIS
LIN {X 57.9846,Y 33.9883,Z 75,A 24.002,B 24.8794,C -2.5344,E1 25.1384,E2 60.1432} C_DIS
LIN {X 60.1584,Y 29.9723,Z 75,A 19.9958,B 24.8807,C -2.5209,E1 25.1437,E2 64.1602} C_DIS
LIN {X 62.0508,Y 25.8275,Z 75,A 15.8924,B 24.8823,C -2.5042,E1 25.1484,E2 68.2807} C_DIS
LIN {X 63.2863,Y 22.6356,Z 75,A 12.7933,B 24.8835,C -2.491,E1 25.1514,E2 71.3937} C_DIS
LIN {X 64.407,Y 19.212,Z 75,A 9.7635,B 24.8843,C -2.483,E1 25.1539,E2 74.4252} C_DIS
LIN {X 65.6286,Y 14.5009,Z 75,A 5.2905,B 24.8862,C -2.4619,E1 25.1568,E2 78.9221} C_DIS
LIN {X 66.6261,Y 8.8529,Z 75,A 1.3444,B 24.8853,C -2.4718,E1 25.1585,E2 82.8218} C_DIS
LIN {X 66.8381,Y 7.0736,Z 75,A -0.5439,B 24.8867,C -2.4574,E1 25.1591,E2 84.7329} C_DIS
LIN {X 67.1832,Y 1.9447,Z 75,A -5.401,B 24.8891,C -2.431,E1 25.1598,E2 89.6235} C_DIS
LIN {X 67.1544,Y -2.7662,Z 75,A -9.1248,B 24.8895,C -2.426,E1 25.1595,E2 93.337} C_DIS
LIN {X 66.9097,Y -6.3629,Z 75,A -11.7536,B 24.8894,C -2.4281,E1 25.1589,E2 95.9453} C_DIS
LIN {X 66.2328,Y -11.4326,Z 75,A -15.9698,B 24.8903,C -2.4181,E1 25.1573,E2 100.1603} C_DIS
LIN {X 65.5763,Y -14.7397,Z 75,A -19.0548,B 24.8916,C -2.4034,E1 25.1555,E2 103.2619} C_DIS
LIN {X 64.8137,Y -17.7937,Z 75,A -22.2697,B 24.8936,C -2.3809,E1 25.1531,E2 106.5114} C_DIS
LIN {X 63.6394,Y -21.6196,Z 75,A -24.8379,B 24.8926,C -2.3928,E1 25.151,E2 109.037} C_DIS
LIN {X 62.6919,Y -24.2322,Z 75,A -27.4702,B 24.8938,C -2.3786,E1 25.1484,E2 111.6883} C_DIS
LIN {X 61.4055,Y -27.3274,Z 75,A -30.3936,B 24.8948,C -2.3683,E1 25.1452,E2 114.6201} C_DIS
LIN {X 60.2163,Y -29.8556,Z 75,A -32.3843,B 24.8945,C -2.3716,E1 25.1428,E2 116.5922} C_DIS
LIN {X 58.7633,Y -32.623,Z 75,A -35.6313,B 24.8965,C -2.3485,E1 25.1384,E2 119.8767} C_DIS
LIN {X 57.3211,Y -35.0956,Z 75,A -37.7749,B 24.8965,C -2.3494,E1 25.1353,E2 122.0073} C_DIS
LIN {X 55.2314,Y -38.2996,Z 75,A -41.0573,B 24.8973,C -2.3398,E1 25.1302,E2 125.2959} C_DIS
LIN {X 53.0743,Y -41.2358,Z 75,A -44.4245,B 24.8986,C -2.3248,E1 25.1245,E2 128.6828} C_DIS
LIN {X 50.4073,Y -44.4586,Z 75,A -48.0545,B 24.8995,C -2.314,E1 25.1179,E2 132.3217} C_DIS
LIN {X 47.3874,Y -47.6638,Z 75,A -51.4537,B 24.8995,C -2.314,E1 25.1113,E2 135.7062} C_DIS
LIN {X 44.3569,Y -50.4961,Z 75,A -54.465,B 24.8991,C -2.3195,E1 25.1051,E2 138.6925} C_DIS
LIN {X 42.6973,Y -51.9077,Z 75,A -57.1224,B 24.9012,C -2.2948,E1 25.0993,E2 141.3981} C_DIS
LIN {X 39.2661,Y -54.5492,Z 75,A -60.5164,B 24.9012,C -2.2948,E1 25.0917,E2 144.7801} C_DIS
LIN {X 35.7921,Y -56.8887,Z 75,A -63.5192,B 24.9005,C -2.3023,E1 25.0848,E2 147.755} C_DIS
LIN {X 34.4351,Y -57.7204,Z 75,A -65.6668,B 24.9025,C -2.2798,E1 25.0795,E2 149.9493} C_DIS
LIN {X 30.189,Y -60.051,Z 75,A -69.1956,B 24.9018,C -2.2879,E1 25.0709,E2 153.4489} C_DIS
LIN {X 28.3661,Y -60.9321,Z 75,A -71.8591,B 24.904,C -2.2619,E1 25.064,E2 156.1673} C_DIS
LIN {X 25.2109,Y -62.304,Z 75,A -74.817,B 24.9044,C -2.2572,E1 25.0564,E2 159.1296} C_DIS
LIN {X 21.8788,Y -63.5518,Z 75,A -77.2541,B 24.9035,C -2.268,E1 25.05,E2 161.5363} C_DIS
LIN {X 16.9239,Y -65.046,Z 75,A -80.9871,B 24.9025,C -2.2799,E1 25.0401,E2 165.2346} C_DIS
LIN {X 11.7941,Y -66.1685,Z 75,A -85.8294,B 24.9036,C -2.2669,E1 25.0268,E2 170.1014} C_DIS
LIN {X 6.3821,Y -66.9079,Z 75,A -90.1116,B 24.9031,C -2.273,E1 25.015,E2 174.3656} C_DIS
LIN {X 4.3634,Y -67.0697,Z 75,A -92.7143,B 24.9049,C -2.2513,E1 25.0076,E2 177.0188} C_DIS
LIN {X 0.474,Y -67.2054,Z 75,A -94.6779,B 24.9022,C -2.2827,E1 25.0024,E2 178.9074} C_DIS
Enddeposition()
LIN {X 0.474,Y -67.2054,Z 75,A -94.6779,B 24.9022,C -2.2827,E1 25.0024,E2 178.9074} C_DIS
Startdeposition()
$VEL.CP = VEL_PRINT
LIN {X 1.534,Y -66.2949,Z 75,A -93.3952,B 24.9001,C -2.3072,E1 25.0061,E2 177.5669} C_DIS
LIN {X 5.5695,Y -66.0782,Z 75,A -90.3274,B 24.9009,C -2.2984,E1 25.0146,E2 174.521} C_DIS
LIN {X 8.5532,Y -65.7579,Z 75,A -87.2567,B 24.8997,C -2.3116,E1 25.0232,E2 171.4214} C_DIS
LIN {X 11.1736,Y -65.3642,Z 75,A -84.1933,B 24.8979,C -2.3324,E1 25.0317,E2 168.3118} C_DIS
LIN {X 14.8633,Y -64.6247,Z 75,A -81.8761,B 24.8997,C -2.3122,E1 25.0379,E2 166.0456} C_DIS
LIN {X 17.8098,Y -63.8761,Z 75,A -79.2252,B 24.8994,C -2.3155,E1 25.0451,E2 163.3911} C_DIS
LIN {X 22.0738,Y -62.5302,Z 75,A -74.9393,B 24.8981,C -2.3308,E1 25.0565,E2 159.0771} C_DIS
LIN {X 26.6209,Y -60.7339,Z 75,A -70.924,B 24.8981,C -2.3315,E1 25.0668,E2 155.0695} C_DIS
LIN {X 29.5736,Y -59.3522,Z 75,A -67.8729,B 24.8971,C -2.342,E1 25.0745,E2 152.0017} C_DIS
LIN {X 34.3451,Y -56.7247,Z 75,A -63.676,B 24.8975,C -2.3373,E1 25.0846,E2 147.8286} C_DIS
LIN {X 38.7371,Y -53.8217,Z 75,A -59.43,B 24.8975,C -2.3384,E1 25.0944,E2 143.5943} C_DIS
LIN {X 42.6059,Y -50.8142,Z 75,A -55.242,B 24.8967,C -2.3462,E1 25.1036,E2 139.4032} C_DIS
LIN {X 45.1542,Y -48.562,Z 75,A -51.7722,B 24.8949,C -2.3668,E1 25.1109,E2 135.8987} C_DIS
LIN {X 48.1971,Y -45.5428,Z 75,A -47.7661,B 24.8934,C -2.3838,E1 25.1187,E2 131.8697} C_DIS
LIN {X 50.4977,Y -42.9796,Z 75,A -44.4798,B 24.8919,C -2.3996,E1 25.1247,E2 128.5609} C_DIS
LIN {X 52.8219,Y -40.0883,Z 75,A -42.3025,B 24.8936,C -2.3807,E1 25.1283,E2 126.4384} C_DIS
LIN {X 55.86,Y -35.7342,Z 75,A -37.6277,B 24.8923,C -2.3956,E1 25.1357,E2 121.7516} C_DIS
LIN {X 57.022,Y -33.8492,Z 75,A -35.6228,B 24.8916,C -2.4035,E1 25.1386,E2 119.7384} C_DIS
LIN {X 59.0924,Y -30.0892,Z 75,A -32.2815,B 24.8916,C -2.4044,E1 25.143,E2 116.4124} C_DIS
LIN {X 60.5201,Y -27.1036,Z 75,A -28.9541,B 24.8896,C -2.4254,E1 25.1469,E2 113.0534} C_DIS
LIN {X 61.8197,Y -23.9929,Z 75,A -26.3664,B 24.8896,C -2.4254,E1 25.1496,E2 110.4798} C_DIS
LIN {X 62.7467,Y -21.4518,Z 75,A -24.005,B 24.8889,C -2.4333,E1 25.1518,E2 108.1133} C_DIS
LIN {X 63.5073,Y -19.0825,Z 75,A -21.9232,B 24.8884,C -2.4381,E1 25.1535,E2 106.0319} C_DIS
LIN {X 64.2316,Y -16.4792,Z 75,A -19.6048,B 24.8878,C -2.445,E1 25.1552,E2 103.7106} C_DIS
LIN {X 64.8738,Y -13.7408,Z 75,A -17.4115,B 24.8877,C -2.4462,E1 25.1565,E2 101.5271} C_DIS
LIN {X 65.3807,Y -11.0746,Z 75,A -14.6862,B 24.8861,C -2.4638,E1 25.1579,E2 98.7761} C_DIS
LIN {X 65.9441,Y -6.9744,Z 75,A -11.5092,B 24.8861,C -2.4645,E1 25.159,E2 95.6164} C_DIS
LIN {X 66.182,Y -4.1441,Z 75,A -8.7975,B 24.8846,C -2.4792,E1 25.1596,E2 92.886} C_DIS
LIN {X 66.2987,Y -1.3272,Z 75,A -6.4839,B 24.8842,C -2.4836,E1 25.1598,E2 90.5757} C_DIS
LIN {X 66.278,Y 2.1206,Z 75,A -3.0864,B 24.8823,C -2.5043,E1 25.1596,E2 87.1496} C_DIS
LIN {X 66.0352,Y 6.0516,Z 75,A 0.0547,B 24.8819,C -2.5079,E1 25.1589,E2 84.0185} C_DIS
LIN {X 65.7437,Y 8.6627,Z 75,A 2.7472,B 24.8802,C -2.5263,E1 25.1579,E2 81.2984} C_DIS
LIN {X 64.8632,Y 13.7894,Z 75,A 6.6839,B 24.8803,C -2.5251,E1 25.1559,E2 77.3875} C_DIS
LIN {X 63.9156,Y 17.664,Z 75,A 10.1217,B 24.8793,C -2.5353,E1 25.1535,E2 73.9455} C_DIS
LIN {X 63.1064,Y 20.3678,Z 75,A 12.5906,B 24.8786,C -2.5433,E1 25.1514,E2 71.4716} C_DIS
LIN {X 62.0456,Y 23.4013,Z 75,A 15.1073,B 24.8785,C -2.5445,E1 25.1491,E2 68.9662} C_DIS
LIN {X 60.6062,Y 26.9087,Z 75,A 18.8072,B 24.8765,C -2.565,E1 25.145,E2 65.2382} C_DIS
LIN {X 59.4896,Y 29.2965,Z 75,A 21.2901,B 24.8754,C -2.5767,E1 25.1419,E2 62.7409} C_DIS
LIN {X 57.6795,Y 32.718,Z 75,A 23.8068,B 24.8766,C -2.5639,E1 25.1386,E2 60.2677} C_DIS
LIN {X 55.6931,Y 35.9942,Z 75,A 27.4188,B 24.875,C -2.5803,E1 25.1333,E2 56.6352} C_DIS
LIN {X 53.9969,Y 38.4915,Z 75,A 29.7685,B 24.875,C -2.5801,E1 25.1295,E2 54.2975} C_DIS
LIN {X 51.4975,Y 41.7765,Z 75,A 33.1915,B 24.8746,C -2.5848,E1 25.1237,E2 50.8795} C_DIS
LIN {X 49.3974,Y 44.2398,Z 75,A 36.3586,B 24.873,C -2.6007,E1 25.1179,E2 47.6893} C_DIS
LIN {X 48,Y 45.7537,Z 75,A 38.5427,B 24.8716,C -2.6149,E1 25.1136,E2 45.481} C_DIS
LIN {X 45.6688,Y 48.0805,Z 75,A 41.3255,B 24.8712,C -2.6191,E1 25.108,E2 42.6999} C_DIS
LIN {X 42.6508,Y 50.7769,Z 75,A 44.8683,B 24.8704,C -2.6269,E1 25.1005,E2 39.1522} C_DIS
LIN {X 40.425,Y 52.5651,Z 75,A 47.8292,B 24.8687,C -2.6438,E1 25.0939,E2 36.162} C_DIS
LIN {X 37.3135,Y 54.8178,Z 75,A 50.1652,B 24.8707,C -2.6244,E1 25.0887,E2 33.88} C_DIS
LIN {X 34.7403,Y 56.4845,Z 75,A 52.8437,B 24.8702,C -2.6292,E1 25.0823,E2 31.1989} C_DIS
LIN {X 31.993,Y 58.0849,Z 75,A 55.5958,B 24.8698,C -2.6331,E1 25.0756,E2 28.4457} C_DIS
LIN {X 29.2046,Y 59.5351,Z 75,A 58.4895,B 24.869,C -2.6409,E1 25.0684,E2 25.5414} C_DIS
LIN {X 26.9526,Y 60.5881,Z 75,A 60.3588,B 24.8695,C -2.6365,E1 25.0637,E2 23.6873} C_DIS
LIN {X 23.933,Y 61.8428,Z 75,A 63.6635,B 24.868,C -2.651,E1 25.055,E2 20.3555} C_DIS
LIN {X 20.2197,Y 63.1543,Z 75,A 66.6792,B 24.8687,C -2.6443,E1 25.0471,E2 17.3614} C_DIS
LIN {X 17.9329,Y 63.8412,Z 75,A 68.9496,B 24.8681,C -2.6507,E1 25.041,E2 15.0796} C_DIS
LIN {X 12.9239,Y 65.0414,Z 75,A 73.1907,B 24.8683,C -2.6479,E1 25.0294,E2 10.8508} C_DIS
LIN {X 10.3057,Y 65.5064,Z 75,A 76.3702,B 24.8662,C -2.6696,E1 25.0205,E2 7.6228} C_DIS
LIN {X 6.5122,Y 65.9925,Z 75,A 79.2393,B 24.8672,C -2.6597,E1 25.0126,E2 4.7792} C_DIS
LIN {X 1.387,Y 66.2976,Z 75,A 83.0217,B 24.8687,C -2.6442,E1 25.0022,E2 1.0348} C_DIS
LIN {X -0.8182,Y 66.3064,Z 75,A 85.163,B 24.8682,C -2.6493,E1 24.9962,E2 -1.1185} C_DIS
LIN {X -4.2738,Y 66.1743,Z 75,A 88.0915,B 24.8685,C -2.6468,E1 24.988,E2 -4.042} C_DIS
LIN {X -8.9644,Y 65.7042,Z 75,A 92.1234,B 24.8688,C -2.6436,E1 24.9769,E2 -8.0688} C_DIS
LIN {X -13.0096,Y 65.024,Z 75,A 95.8686,B 24.8686,C -2.6455,E1 24.9665,E2 -11.8222} C_DIS
LIN {X -17.4789,Y 63.9671,Z 75,A 99.7007,B 24.8693,C -2.6386,E1 24.9562,E2 -15.6435} C_DIS
LIN {X -20.1007,Y 63.1928,Z 75,A 102.1815,B 24.8693,C -2.6386,E1 24.9496,E2 -18.1285} C_DIS
LIN {X -24.3376,Y 61.6843,Z 75,A 105.8128,B 24.8703,C -2.628,E1 24.9401,E2 -21.7421} C_DIS
LIN {X -26.1255,Y 60.9499,Z 75,A 107.9422,B 24.8696,C -2.6357,E1 24.9346,E2 -23.8947} C_DIS
LIN {X -29.4497,Y 59.4136,Z 75,A 110.7991,B 24.8707,C -2.6241,E1 24.9274,E2 -26.7314} C_DIS
LIN {X -32.348,Y 57.8867,Z 75,A 114.5448,B 24.8692,C -2.6392,E1 24.9182,E2 -30.5237} C_DIS
LIN {X -35.5566,Y 55.974,Z 75,A 116.7593,B 24.872,C -2.6114,E1 24.9131,E2 -32.6789} C_DIS
LIN {X -38.9614,Y 53.6587,Z 75,A 120.3115,B 24.8727,C -2.6043,E1 24.9049,E2 -36.2263} C_DIS
LIN {X -41.2517,Y 51.9184,Z 75,A 123.7776,B 24.8711,C -2.6199,E1 24.8972,E2 -39.7424} C_DIS
LIN {X -43.977,Y 49.6327,Z 75,A 126.0256,B 24.8735,C -2.5956,E1 24.8926,E2 -41.9411} C_DIS
LIN {X -46.1007,Y 47.6655,Z 75,A 128.8511,B 24.8735,C -2.5966,E1 24.8868,E2 -44.7807} C_DIS
LIN {X -48.4085,Y 45.32,Z 75,A 131.1722,B 24.8751,C -2.5788,E1 24.8824,E2 -47.0694} C_DIS
LIN {X -51.2663,Y 42.0617,Z 75,A 134.9769,B 24.8759,C -2.5706,E1 24.8755,E2 -50.8717} C_DIS
LIN {X -53.7604,Y 38.8214,Z 75,A 138.7147,B 24.8764,C -2.5654,E1 24.8692,E2 -54.6151} C_DIS
LIN {X -55.8452,Y 35.7573,Z 75,A 142.3807,B 24.8764,C -2.5662,E1 24.8635,E2 -58.3012} C_DIS
LIN {X -58.7522,Y 30.7485,Z 75,A 147.3072,B 24.8779,C -2.5502,E1 24.8568,E2 -63.2155} C_DIS
LIN {X -60.5222,Y 27.0989,Z 75,A 150.8566,B 24.8788,C -2.5408,E1 24.8527,E2 -66.7618} C_DIS
LIN {X -62.1476,Y 23.1319,Z 75,A 154.3354,B 24.8803,C -2.525,E1 24.8492,E2 -70.2223} C_DIS
LIN {X -63.1797,Y 20.1414,Z 75,A 156.8126,B 24.8816,C -2.5115,E1 24.847,E2 -72.6814} C_DIS
LIN {X -63.7959,Y 18.0926,Z 75,A 159.1605,B 24.8812,C -2.5158,E1 24.8452,E2 -75.0533} C_DIS
LIN {X -64.5074,Y 15.3684,Z 75,A 161.4445,B 24.8822,C -2.5052,E1 24.8437,E2 -77.3253} C_DIS
LIN {X -65.3545,Y 11.2311,Z 75,A 165.052,B 24.8834,C -2.4929,E1 24.8418,E2 -80.9246} C_DIS
LIN {X -65.807,Y 8.1743,Z 75,A 167.6972,B 24.8842,C -2.4839,E1 24.8408,E2 -83.5643} C_DIS
LIN {X -66.1024,Y 5.2662,Z 75,A 170.6017,B 24.8842,C -2.4836,E1 24.8401,E2 -86.4855} C_DIS
LIN {X -66.3085,Y -0.7668,Z 75,A 175.5273,B 24.8863,C -2.4612,E1 24.8398,E2 -91.3871} C_DIS
LIN {X -65.9322,Y -7.088,Z 75,A -179.3869,B 24.8886,C -2.4362,E1 24.8408,E2 -96.4437} C_DIS
LIN {X -65.4997,Y -10.3488,Z 75,A -176.127,B 24.8886,C -2.4358,E1 24.8421,E2 -99.7221} C_DIS
LIN {X -64.9661,Y -13.2918,Z 75,A -173.644,B 24.8896,C -2.4258,E1 24.8434,E2 -102.1959} C_DIS
LIN {X -64.5597,Y -15.1444,Z 75,A -171.674,B 24.8894,C -2.4276,E1 24.8446,E2 -104.1818} C_DIS
LIN {X -63.5201,Y -19.0394,Z 75,A -168.3693,B 24.8907,C -2.4135,E1 24.8471,E2 -107.472} C_DIS
LIN {X -62.6179,Y -21.8239,Z 75,A -165.7098,B 24.8911,C -2.4088,E1 24.8495,E2 -110.1354} C_DIS
LIN {X -61.3372,Y -25.1986,Z 75,A -162.5761,B 24.8919,C -2.4002,E1 24.8527,E2 -113.2661} C_DIS
LIN {X -59.8556,Y -28.5413,Z 75,A -158.6178,B 24.8912,C -2.4081,E1 24.8575,E2 -117.2647} C_DIS
LIN {X -58.1728,Y -31.8315,Z 75,A -156.1199,B 24.8933,C -2.3849,E1 24.8607,E2 -119.7206} C_DIS
LIN {X -56.4636,Y -34.7747,Z 75,A -153.3744,B 24.8943,C -2.3732,E1 24.8646,E2 -122.4522} C_DIS
LIN {X -54.9071,Y -37.1816,Z 75,A -150.8775,B 24.8948,C -2.3674,E1 24.8685,E2 -124.9478} C_DIS
LIN {X -53.1194,Y -39.6941,Z 75,A -148.2173,B 24.8954,C -2.3608,E1 24.8728,E2 -127.6052} C_DIS
LIN {X -50.7122,Y -42.7279,Z 75,A -144.611,B 24.8956,C -2.3586,E1 24.8792,E2 -131.2229} C_DIS
LIN {X -48.0798,Y -45.6695,Z 75,A -141.1318,B 24.8961,C -2.3526,E1 24.8858,E2 -134.7032} C_DIS
LIN {X -45.9474,Y -47.8133,Z 75,A -138.2771,B 24.8961,C -2.3526,E1 24.8916,E2 -137.5696} C_DIS
LIN {X -42.6925,Y -50.7423,Z 75,A -134.4912,B 24.8968,C -2.3454,E1 24.8996,E2 -141.3532} C_DIS
LIN {X -39.8447,Y -53.0063,Z 75,A -132.0974,B 24.8987,C -2.3235,E1 24.9048,E2 -143.7036} C_DIS
LIN {X -36.6951,Y -55.2339,Z 75,A -128.5111,B 24.8987,C -2.3235,E1 24.913,E2 -147.3024} C_DIS
LIN {X -34.5094,Y -56.6248,Z 75,A -126.2195,B 24.8989,C -2.3215,E1 24.9184,E2 -149.5961} C_DIS
LIN {X -30.8898,Y -58.6778,Z 75,A -122.7928,B 24.8996,C -2.3129,E1 24.9268,E2 -153.0122} C_DIS
LIN {X -29.2274,Y -59.5236,Z 75,A -120.6167,B 24.8987,C -2.3236,E1 24.9323,E2 -155.2196} C_DIS
LIN {X -24.5251,Y -61.6106,Z 75,A -116.5596,B 24.8999,C -2.3102,E1 24.9427,E2 -159.2542} C_DIS
LIN {X -21.7347,Y -62.6492,Z 75,A -114.2225,B 24.9005,C -2.3027,E1 24.9488,E2 -161.578} C_DIS
LIN {X -18.9323,Y -63.5518,Z 75,A -110.7351,B 24.8988,C -2.3226,E1 24.9582,E2 -165.1188} C_DIS
LIN {X -14.4323,Y -64.723,Z 75,A -107.6987,B 24.901,C -2.2977,E1 24.9663,E2 -168.1001} C_DIS
LIN {X -11.6162,Y -65.2866,Z 75,A -104.7577,B 24.9001,C -2.3074,E1 24.9745,E2 -171.0675} C_DIS
LIN {X -9.1072,Y -65.6839,Z 75,A -102.5056,B 24.9001,C -2.3083,E1 24.9807,E2 -173.3235} C_DIS
LIN {X -5.3611,Y -66.0948,Z 75,A -99.1958,B 24.8999,C -2.3093,E1 24.9899,E2 -176.6375} C_DIS
LIN {X -1.1162,Y -66.3021,Z 75,A -95.8412,B 24.9006,C -2.3022,E1 24.9992,E2 -179.9757} C_DIS
LIN {X -1.1162,Y -66.3021,Z 75,A -95.8412,B 24.9006,C -2.3022,E1 24.9992,E2 -179.9757} C_DIS
Enddeposition()
LIN {X 0.4557,Y -65.4055,Z 75,A -95.0448,B 24.9003,C -2.3048,E1 25.0015,E2 -180.7784} C_DIS
Startdeposition()
$VEL.CP = VEL_PRINT
LIN {X -2.252,Y -65.3741,Z 75,A -97.8555,B 24.9013,C -2.2942,E1 24.9936,E2 -177.9421} C_DIS
LIN {X -4.5116,Y -65.2567,Z 75,A -100.9922,B 24.9035,C -2.268,E1 24.9847,E2 -174.742} C_DIS
LIN {X -8.2936,Y -64.8846,Z 75,A -103.2061,B 24.9013,C -2.2935,E1 24.9787,E2 -172.5873} C_DIS
LIN {X -12.2777,Y -64.2499,Z 75,A -106.6642,B 24.9011,C -2.2963,E1 24.9692,E2 -169.1325} C_DIS
LIN {X -14.7071,Y -63.7376,Z 75,A -109.0247,B 24.9013,C -2.2931,E1 24.9627,E2 -166.7615} C_DIS
LIN {X -18.2808,Y -62.8067,Z 75,A -112.2767,B 24.9013,C -2.2947,E1 24.9539,E2 -163.5083} C_DIS
LIN {X -20.0941,Y -62.2496,Z 75,A -114.0138,B 24.9013,C -2.2943,E1 24.9493,E2 -161.767} C_DIS
LIN {X -22.9576,Y -61.2518,Z 75,A -116.6121,B 24.9009,C -2.2978,E1 24.9425,E2 -159.1721} C_DIS
LIN {X -26.7167,Y -59.7079,Z 75,A -120.4686,B 24.9012,C -2.2951,E1 24.9325,E2 -155.3} C_DIS
LIN {X -29.7863,Y -58.2371,Z 75,A -123.7947,B 24.9015,C -2.2913,E1 24.9242,E2 -151.9562} C_DIS
LIN {X -33.5838,Y -56.1341,Z 75,A -126.9479,B 24.8999,C -2.3104,E1 24.9166,E2 -148.839} C_DIS
LIN {X -35.8973,Y -54.6826,Z 75,A -129.7476,B 24.9003,C -2.3054,E1 24.91,E2 -146.0185} C_DIS
LIN {X -39.2099,Y -52.3582,Z 75,A -133.3008,B 24.8998,C -2.3112,E1 24.902,E2 -142.4666} C_DIS
LIN {X -42.0858,Y -50.077,Z 75,A -135.9802,B 24.8983,C -2.3282,E1 24.8963,E2 -139.8176} C_DIS
LIN {X -45.4402,Y -47.053,Z 75,A -139.9516,B 24.8976,C -2.3357,E1 24.8881,E2 -135.848} C_DIS
LIN {X -47.4359,Y -45.0413,Z 75,A -142.6491,B 24.8976,C -2.3365,E1 24.8828,E2 -133.1409} C_DIS
LIN {X -50.0825,Y -42.0791,Z 75,A -146.1959,B 24.897,C -2.3429,E1 24.8763,E2 -129.5933} C_DIS
LIN {X -52.105,Y -39.5469,Z 75,A -148.8752,B 24.8961,C -2.3528,E1 24.8717,E2 -126.9251} C_DIS
LIN {X -54.0904,Y -36.7837,Z 75,A -151.9004,B 24.8956,C -2.3592,E1 24.8668,E2 -123.9003} C_DIS
LIN {X -55.6567,Y -34.369,Z 75,A -154.5256,B 24.8952,C -2.3636,E1 24.8629,E2 -121.2722} C_DIS
LIN {X -57.1986,Y -31.7355,Z 75,A -157.6716,B 24.8954,C -2.3613,E1 24.8585,E2 -118.1042} C_DIS
LIN {X -58.7644,Y -28.7344,Z 75,A -160.2735,B 24.894,C -2.3765,E1 24.8553,E2 -115.5247} C_DIS
LIN {X -60.0669,Y -25.9003,Z 75,A -163.5276,B 24.8942,C -2.3739,E1 24.8516,E2 -112.2466} C_DIS
LIN {X -61.7308,Y -21.6354,Z 75,A -167.2475,B 24.8927,C -2.3912,E1 24.848,E2 -108.5469} C_DIS
LIN {X -62.7856,Y -18.3527,Z 75,A -170.0812,B 24.8916,C -2.4038,E1 24.8457,E2 -105.727} C_DIS
LIN {X -63.5334,Y -15.5661,Z 75,A -172.4532,B 24.8906,C -2.4144,E1 24.8441,E2 -103.3665} C_DIS
LIN {X -64.1677,Y -12.7046,Z 75,A -175.2732,B 24.8903,C -2.4173,E1 24.8425,E2 -100.5368} C_DIS
LIN {X -64.7087,Y -9.5766,Z 75,A -178.1962,B 24.8898,C -2.4232,E1 24.8412,E2 -97.6103} C_DIS
LIN {X -65.0464,Y -6.9109,Z 75,A 178.9711,B 24.89,C -2.4213,E1 24.8403,E2 -94.7563} C_DIS
LIN {X -65.3449,Y -2.9766,Z 75,A 176.1468,B 24.8879,C -2.4443,E1 24.8399,E2 -91.97} C_DIS
LIN {X -65.4141,Y 0.1034,Z 75,A 172.9518,B 24.8879,C -2.4433,E1 24.8399,E2 -88.7532} C_DIS
LIN {X -65.2705,Y 4.3084,Z 75,A 169.7465,B 24.886,C -2.4642,E1 24.8403,E2 -85.5786} C_DIS
LIN {X -65.0051,Y 7.2957,Z 75,A 167.0913,B 24.8853,C -2.4719,E1 24.841,E2 -82.9261} C_DIS
LIN {X -64.6005,Y 10.2785,Z 75,A 164.4159,B 24.8846,C -2.4795,E1 24.8421,E2 -80.2528} C_DIS
LIN {X -63.9165,Y 13.9092,Z 75,A 161.3401,B 24.8834,C -2.4928,E1 24.8437,E2 -77.1906} C_DIS
LIN {X -63.4921,Y 15.7351,Z 75,A 159.4871,B 24.8833,C -2.4938,E1 24.845,E2 -75.3292} C_DIS
LIN {X -62.2944,Y 19.9557,Z 75,A 155.8786,B 24.8817,C -2.5103,E1 24.8478,E2 -71.7392} C_DIS
LIN {X -61.5472,Y 22.1541,Z 75,A 153.5815,B 24.8817,C -2.5113,E1 24.8499,E2 -69.4316} C_DIS
LIN {X -60.4371,Y 25.0259,Z 75,A 150.8328,B 24.8809,C -2.5184,E1 24.8528,E2 -66.6845} C_DIS
LIN {X -59.1036,Y 28.0297,Z 75,A 147.2718,B 24.8814,C -2.5138,E1 24.857,E2 -63.0929} C_DIS
LIN {X -56.5753,Y 32.8345,Z 75,A 143.5784,B 24.8781,C -2.5481,E1 24.8619,E2 -59.462} C_DIS
LIN {X -54.1043,Y 36.7631,Z 75,A 139.2799,B 24.8775,C -2.5548,E1 24.8683,E2 -55.1577} C_DIS
LIN {X -51.4416,Y 40.4053,Z 75,A 135.1722,B 24.8768,C -2.5622,E1 24.8752,E2 -51.0479} C_DIS
LIN {X -47.643,Y 44.8211,Z 75,A 130.2495,B 24.8752,C -2.5786,E1 24.8842,E2 -46.1422} C_DIS
LIN {X -46.3523,Y 46.1554,Z 75,A 128.1066,B 24.8758,C -2.5721,E1 24.8884,E2 -43.9747} C_DIS
LIN {X -44.5125,Y 47.933,Z 75,A 126.0775,B 24.8749,C -2.5815,E1 24.8925,E2 -41.9596} C_DIS
LIN {X -41.2576,Y 50.7603,Z 75,A 121.8922,B 24.8749,C -2.5815,E1 24.9015,E2 -37.7584} C_DIS
LIN {X -36.1136,Y 54.54,Z 75,A 116.756,B 24.8729,C -2.602,E1 24.9131,E2 -32.6531} C_DIS
LIN {X -32.5465,Y 56.7408,Z 75,A 112.9115,B 24.8726,C -2.605,E1 24.9223,E2 -28.8041} C_DIS
LIN {X -30.0126,Y 58.1215,Z 75,A 110.2718,B 24.8724,C -2.6068,E1 24.9288,E2 -26.1615} C_DIS
LIN {X -26.1989,Y 59.9367,Z 75,A 106.9999,B 24.871,C -2.6214,E1 24.9371,E2 -22.916} C_DIS
LIN {X -21.6743,Y 61.7172,Z 75,A 102.6422,B 24.8706,C -2.6249,E1 24.9484,E2 -18.5574} C_DIS
LIN {X -18.9595,Y 62.6056,Z 75,A 99.8852,B 24.8709,C -2.6223,E1 24.9558,E2 -15.7894} C_DIS
LIN {X -15.3491,Y 63.5863,Z 75,A 96.2194,B 24.8714,C -2.6172,E1 24.9658,E2 -12.1061} C_DIS
LIN {X -11.4203,Y 64.408,Z 75,A 93.1567,B 24.8702,C -2.6297,E1 24.9741,E2 -9.0699} C_DIS
LIN {X -8.5652,Y 64.8494,Z 75,A 89.7973,B 24.8718,C -2.6133,E1 24.9835,E2 -5.6689} C_DIS
LIN {X -5.0869,Y 65.2145,Z 75,A 87.7974,B 24.8693,C -2.638,E1 24.9889,E2 -3.7267} C_DIS
LIN {X -2.2076,Y 65.3755,Z 75,A 84.8605,B 24.8702,C -2.6297,E1 24.9972,E2 -0.7695} C_DIS
LIN {X 1.2867,Y 65.3998,Z 75,A 80.9802,B 24.8719,C -2.6121,E1 25.0081,E2 3.1521} C_DIS
LIN {X 5.1663,Y 65.2081,Z 75,A 78.7553,B 24.8693,C -2.6383,E1 25.0141,E2 5.3139} C_DIS
LIN {X 8.9888,Y 64.7922,Z 75,A 75.2971,B 24.8696,C -2.6356,E1 25.0237,E2 8.7758} C_DIS
LIN {X 11.7355,Y 64.3513,Z 75,A 72.722,B 24.87,C -2.6317,E1 25.0308,E2 11.3577} C_DIS
LIN {X 15.2288,Y 63.6156,Z 75,A 69.6779,B 24.87,C -2.632,E1 25.0391,E2 14.3968} C_DIS
LIN {X 17.6183,Y 62.9955,Z 75,A 67.548,B 24.87,C -2.6314,E1 25.0448,E2 16.5248} C_DIS
LIN {X 20.2908,Y 62.186,Z 75,A 65.053,B 24.8703,C -2.6284,E1 25.0515,E2 19.0224} C_DIS
LIN {X 24.1826,Y 60.7789,Z 75,A 60.9346,B 24.8718,C -2.6134,E1 25.0623,E2 23.1673} C_DIS
LIN {X 29.679,Y 58.292,Z 75,A 56.3232,B 24.8708,C -2.6232,E1 25.0739,E2 27.7438} C_DIS
LIN {X 31.2307,Y 57.4755,Z 75,A 54.613,B 24.8714,C -2.617,E1 25.0781,E2 29.4638} C_DIS
LIN {X 33.9005,Y 55.9424,Z 75,A 51.985,B 24.8716,C -2.6148,E1 25.0844,E2 32.089} C_DIS
LIN {X 36.3761,Y 54.3663,Z 75,A 49.3607,B 24.8722,C -2.6095,E1 25.0906,E2 34.7173} C_DIS
LIN {X 39.8669,Y 51.8596,Z 75,A 45.4223,B 24.8732,C -2.5988,E1 25.0995,E2 38.667} C_DIS
LIN {X 42.6166,Y 49.6254,Z 75,A 42.5439,B 24.8732,C -2.5985,E1 25.1056,E2 41.535} C_DIS
LIN {X 44.9463,Y 47.5252,Z 75,A 40.0723,B 24.8732,C -2.5998,E1 25.1107,E2 43.9935} C_DIS
LIN {X 46.7988,Y 45.7034,Z 75,A 37.8345,B 24.8735,C -2.596,E1 25.1151,E2 46.2309} C_DIS
LIN {X 49.1571,Y 43.1555,Z 75,A 34.3157,B 24.8753,C -2.5774,E1 25.1217,E2 49.778} C_DIS
LIN {X 50.7783,Y 41.2354,Z 75,A 31.8079,B 24.8765,C -2.5647,E1 25.1262,E2 52.3044} C_DIS
LIN {X 53.3359,Y 37.8694,Z 75,A 28.6168,B 24.8762,C -2.5684,E1 25.1314,E2 55.4712} C_DIS
LIN {X 55.0387,Y 35.3487,Z 75,A 25.7189,B 24.8774,C -2.5558,E1 25.1359,E2 58.3844} C_DIS
LIN {X 57.0179,Y 32.0591,Z 75,A 21.9394,B 24.8792,C -2.5365,E1 25.1412,E2 62.1901} C_DIS
LIN {X 59.1004,Y 28.0356,Z 75,A 17.7802,B 24.8807,C -2.5207,E1 25.1463,E2 66.3644} C_DIS
LIN {X 60.5872,Y 24.6573,Z 75,A 16.1026,B 24.8778,C -2.5512,E1 25.148,E2 67.9607} C_DIS
LIN {X 61.3297,Y 22.7505,Z 75,A 13.6873,B 24.8798,C -2.53,E1 25.1505,E2 70.4127} C_DIS
LIN {X 62.4958,Y 19.3147,Z 75,A 10.1119,B 24.8817,C -2.5104,E1 25.1536,E2 74.014} C_DIS
LIN {X 63.4357,Y 15.9628,Z 75,A 7.4866,B 24.8815,C -2.5121,E1 25.1554,E2 76.6202} C_DIS
LIN {X 64.1244,Y 12.9192,Z 75,A 4.4887,B 24.883,C -2.497,E1 25.1572,E2 79.6365} C_DIS
LIN {X 64.846,Y 8.5917,Z 75,A 1.445,B 24.8821,C -2.5058,E1 25.1585,E2 82.6415} C_DIS
LIN {X 65.1517,Y 5.8372,Z 75,A -1.7309,B 24.8847,C -2.4788,E1 25.1594,E2 85.8624} C_DIS
LIN {X 65.3728,Y 2.2966,Z 75,A -4.4263,B 24.8846,C -2.4796,E1 25.1597,E2 88.5398} C_DIS
LIN {X 65.4089,Y -0.724,Z 75,A -7.1688,B 24.8856,C -2.4687,E1 25.1597,E2 91.2917} C_DIS
LIN {X 65.3013,Y -3.8174,Z 75,A -9.9238,B 24.8865,C -2.459,E1 25.1594,E2 94.0533} C_DIS
LIN {X 65.0396,Y -6.9761,Z 75,A -13.4324,B 24.8891,C -2.4313,E1 25.1584,E2 97.6066} C_DIS
LIN {X 64.5652,Y -10.4981,Z 75,A -15.6663,B 24.8879,C -2.4441,E1 25.1574,E2 99.797} C_DIS
LIN {X 64.0411,Y -13.3247,Z 75,A -18.1719,B 24.8886,C -2.4365,E1 25.1561,E2 102.306} C_DIS
LIN {X 63.3827,Y -16.1688,Z 75,A -20.6839,B 24.8892,C -2.4297,E1 25.1544,E2 104.8196} C_DIS
LIN {X 62.6563,Y -18.7886,Z 75,A -23.1653,B 24.8901,C -2.4197,E1 25.1525,E2 107.3103} C_DIS
LIN {X 61.256,Y -22.9461,Z 75,A -26.6518,B 24.8904,C -2.4172,E1 25.1493,E2 110.7832} C_DIS
LIN {X 60.6377,Y -24.5331,Z 75,A -28.8448,B 24.8924,C -2.3945,E1 25.147,E2 113.0176} C_DIS
LIN {X 58.4299,Y -29.4091,Z 75,A -32.7547,B 24.8918,C -2.4007,E1 25.1424,E2 116.8918} C_DIS
LIN {X 56.7187,Y -32.5849,Z 75,A -36.027,B 24.8929,C -2.3887,E1 25.138,E2 120.1753} C_DIS
LIN {X 55.4343,Y -34.7251,Z 75,A -38.2319,B 24.8935,C -2.3821,E1 25.1348,E2 122.3848} C_DIS
LIN {X 53.7134,Y -37.3317,Z 75,A -40.8853,B 24.894,C -2.3766,E1 25.1306,E2 125.0378} C_DIS
LIN {X 51.8474,Y -39.8828,Z 75,A -44.2137,B 24.8959,C -2.355,E1 25.125,E2 128.4015} C_DIS
LIN {X 49.4569,Y -42.8122,Z 75,A -47.5833,B 24.8968,C -2.345,E1 25.1189,E2 131.7793} C_DIS
LIN {X 46.2431,Y -46.2655,Z 75,A -50.917,B 24.8959,C -2.3551,E1 25.1125,E2 135.0747} C_DIS
LIN {X 43.0953,Y -49.2097,Z 75,A -54.9943,B 24.8974,C -2.3387,E1 25.1041,E2 139.1742} C_DIS
LIN {X 40.0064,Y -51.7521,Z 75,A -58.6236,B 24.8983,C -2.328,E1 25.0962,E2 142.8152} C_DIS
LIN {X 36.5813,Y -54.2273,Z 75,A -61.7113,B 24.8976,C -2.3359,E1 25.0892,E2 145.8736} C_DIS
LIN {X 34.9479,Y -55.2951,Z 75,A -63.8802,B 24.8989,C -2.3212,E1 25.0841,E2 148.0702} C_DIS
LIN {X 31.3187,Y -57.4278,Z 75,A -67.7922,B 24.9,C -2.3092,E1 25.0745,E2 151.999} C_DIS
LIN {X 28.9582,Y -58.6534,Z 75,A -70.3681,B 24.9008,C -2.2994,E1 25.068,E2 154.591} C_DIS
LIN {X 23.9537,Y -60.8688,Z 75,A -74.7565,B 24.9005,C -2.3023,E1 25.0568,E2 158.9623} C_DIS
LIN {X 19.6163,Y -62.4023,Z 75,A -78.3547,B 24.9001,C -2.3077,E1 25.0474,E2 162.5405} C_DIS
LIN {X 17.37,Y -63.0648,Z 75,A -80.673,B 24.9008,C -2.2991,E1 25.0411,E2 164.8755} C_DIS
LIN {X 14.6601,Y -63.7485,Z 75,A -83.614,B 24.902,C -2.285,E1 25.033,E2 167.8456} C_DIS
LIN {X 11.1145,Y -64.4621,Z 75,A -86.1038,B 24.9009,C -2.2985,E1 25.0263,E2 170.3007} C_DIS
LIN {X 6.798,Y -65.0582,Z 75,A -89.6668,B 24.9006,C -2.302,E1 25.0165,E2 173.8523} C_DIS
LIN {X 4.5,Y -65.2575,Z 75,A -92.2195,B 24.9017,C -2.2886,E1 25.0093,E2 176.4356} C_DIS
LIN {X 1.3156,Y -65.3993,Z 75,A -95.0044,B 24.9018,C -2.2878,E1 25.0015,E2 179.2216} C_DIS
LIN {X 1.3156,Y -65.3993,Z 75,A -95.0044,B 24.9018,C -2.2878,E1 25.0015,E2 179.2216} C_DIS
Enddeposition()
LIN {X 0.4637,Y -64.5008,Z 75,A -95.9515,B 24.9008,C -2.2991,E1 24.9989,E2 180.1419} C_DIS
Startdeposition()
$VEL.CP = VEL_PRINT
LIN {X 2.1869,Y -64.4763,Z 75,A -92.2202,B 24.8964,C -2.3503,E1 25.0097,E2 176.2899} C_DIS
LIN {X 6.9686,Y -64.136,Z 75,A -88.648,B 24.8976,C -2.3362,E1 25.0195,E2 172.7531} C_DIS
LIN {X 9.931,Y -63.7441,Z 75,A -85.3406,B 24.8961,C -2.3537,E1 25.0287,E2 169.4073} C_DIS
LIN {X 14.4569,Y -62.8723,Z 75,A -81.9605,B 24.8972,C -2.3401,E1 25.0379,E2 166.0637} C_DIS
LIN {X 17.4181,Y -62.1174,Z 75,A -79.3478,B 24.8972,C -2.3405,E1 25.0449,E2 163.4543} C_DIS
LIN {X 19.8617,Y -61.3795,Z 75,A -77.0886,B 24.897,C -2.3429,E1 25.0509,E2 161.1934} C_DIS
LIN {X 22.4659,Y -60.4761,Z 75,A -74.7336,B 24.897,C -2.3438,E1 25.0571,E2 158.8411} C_DIS
LIN {X 26.4955,Y -58.8211,Z 75,A -70.6935,B 24.8961,C -2.3535,E1 25.0676,E2 154.7874} C_DIS
LIN {X 29.0384,Y -57.6093,Z 75,A -68.2243,B 24.8958,C -2.3567,E1 25.0737,E2 152.3172} C_DIS
LIN {X 32.74,Y -55.5881,Z 75,A -64.5269,B 24.8953,C -2.3621,E1 25.0828,E2 148.618} C_DIS
LIN {X 35.2648,Y -54.0223,Z 75,A -61.9208,B 24.8949,C -2.3662,E1 25.0889,E2 146.0105} C_DIS
LIN {X 37.3038,Y -52.6346,Z 75,A -59.7509,B 24.8946,C -2.3701,E1 25.0939,E2 143.8389} C_DIS
LIN {X 40.1795,Y -50.4737,Z 75,A -56.4701,B 24.8938,C -2.379,E1 25.1012,E2 140.549} C_DIS
LIN {X 42.4555,Y -48.5743,Z 75,A -53.8146,B 24.8932,C -2.3855,E1 25.1068,E2 137.8886} C_DIS
LIN {X 44.5866,Y -46.6265,Z 75,A -50.902,B 24.8919,C -2.4003,E1 25.1128,E2 134.9528} C_DIS
LIN {X 47.9734,Y -43.1335,Z 75,A -47.0177,B 24.8919,C -2.3998,E1 25.1202,E2 131.0868} C_DIS
LIN {X 49.9272,Y -40.857,Z 75,A -44.341,B 24.8913,C -2.4069,E1 25.125,E2 128.4054} C_DIS
LIN {X 51.115,Y -39.3596,Z 75,A -42.274,B 24.89,C -2.421,E1 25.1285,E2 126.315} C_DIS
LIN {X 53.5298,Y -36.0074,Z 75,A -38.9853,B 24.89,C -2.4211,E1 25.1338,E2 123.042} C_DIS
LIN {X 55.148,Y -33.4758,Z 75,A -36.3451,B 24.8894,C -2.4279,E1 25.1377,E2 120.3993} C_DIS
LIN {X 56.4108,Y -31.3015,Z 75,A -33.9546,B 24.8884,C -2.4384,E1 25.141,E2 117.9963} C_DIS
LIN {X 57.9803,Y -28.2905,Z 75,A -31.1079,B 24.888,C -2.4428,E1 25.1445,E2 115.1544} C_DIS
LIN {X 59.9174,Y -23.9157,Z 75,A -27.1681,B 24.8876,C -2.4475,E1 25.1489,E2 111.2251} C_DIS
LIN {X 60.6997,Y -21.8523,Z 75,A -24.9358,B 24.8864,C -2.4605,E1 25.151,E2 108.9744} C_DIS
LIN {X 61.5893,Y -19.2016,Z 75,A -22.641,B 24.8861,C -2.4633,E1 25.153,E2 106.6861} C_DIS
LIN {X 62.2869,Y -16.801,Z 75,A -20.4166,B 24.8855,C -2.4703,E1 25.1547,E2 104.4579} C_DIS
LIN {X 62.8989,Y -14.3418,Z 75,A -18.1493,B 24.8848,C -2.4778,E1 25.1562,E2 102.186} C_DIS
LIN {X 63.4427,Y -11.7062,Z 75,A -15.8324,B 24.8842,C -2.4834,E1 25.1574,E2 99.8694} C_DIS
LIN {X 63.7459,Y -9.9191,Z 75,A -13.9496,B 24.8831,C -2.4956,E1 25.1582,E2 97.9688} C_DIS
LIN {X 64.1778,Y -6.57,Z 75,A -11.1034,B 24.8826,C -2.5011,E1 25.1591,E2 95.1264} C_DIS
LIN {X 64.4112,Y -3.6231,Z 75,A -8.6831,B 24.8823,C -2.5041,E1 25.1596,E2 92.7134} C_DIS
LIN {X 64.5003,Y -1.2844,Z 75,A -6.6462,B 24.8818,C -2.5096,E1 25.1598,E2 90.6756} C_DIS
LIN {X 64.4663,Y 2.4728,Z 75,A -3.0851,B 24.8802,C -2.526,E1 25.1596,E2 87.097} C_DIS
LIN {X 64.2304,Y 6.0333,Z 75,A 0.4403,B 24.8784,C -2.5453,E1 25.1588,E2 83.5469} C_DIS
LIN {X 63.7623,Y 9.8135,Z 75,A 3.7554,B 24.8775,C -2.554,E1 25.1574,E2 80.2308} C_DIS
LIN {X 63.0517,Y 13.6537,Z 75,A 6.8694,B 24.8775,C -2.5553,E1 25.1557,E2 77.1317} C_DIS
LIN {X 62.4138,Y 16.3256,Z 75,A 9.3167,B 24.8767,C -2.5629,E1 25.1541,E2 74.6806} C_DIS
LIN {X 61.5382,Y 19.3662,Z 75,A 11.9985,B 24.8762,C -2.5679,E1 25.1519,E2 72.0023} C_DIS
LIN {X 60.7008,Y 21.8498,Z 75,A 14.3287,B 24.8755,C -2.5748,E1 25.1498,E2 69.6689} C_DIS
LIN {X 59.5324,Y 24.8569,Z 75,A 17.6949,B 24.8735,C -2.5959,E1 25.1462,E2 66.2714} C_DIS
LIN {X 57.7865,Y 28.6818,Z 75,A 20.8944,B 24.8738,C -2.5925,E1 25.1424,E2 63.0972} C_DIS
LIN {X 56.3559,Y 31.3998,Z 75,A 24.1372,B 24.8718,C -2.613,E1 25.138,E2 59.8229} C_DIS
LIN {X 54.0466,Y 35.228,Z 75,A 27.5663,B 24.8722,C -2.6093,E1 25.1329,E2 56.4197} C_DIS
LIN {X 52.3285,Y 37.7328,Z 75,A 30.2844,B 24.8715,C -2.6165,E1 25.1286,E2 53.6979} C_DIS
LIN {X 50.8953,Y 39.6448,Z 75,A 32.4658,B 24.8708,C -2.6231,E1 25.1248,E2 51.5113} C_DIS
LIN {X 48.7746,Y 42.2261,Z 75,A 35.3123,B 24.8704,C -2.6268,E1 25.1197,E2 48.669} C_DIS
LIN {X 46.6894,Y 44.5213,Z 75,A 38.0985,B 24.8698,C -2.6336,E1 25.1144,E2 45.8788} C_DIS
LIN {X 44.4786,Y 46.7305,Z 75,A 40.9079,B 24.8691,C -2.6402,E1 25.1088,E2 43.0657} C_DIS
LIN {X 42.1253,Y 48.8623,Z 75,A 43.6479,B 24.8688,C -2.6437,E1 25.103,E2 40.3282} C_DIS
LIN {X 40.0353,Y 50.5876,Z 75,A 45.8423,B 24.8688,C -2.6429,E1 25.0983,E2 38.144} C_DIS
LIN {X 37.7677,Y 52.3035,Z 75,A 48.5622,B 24.8679,C -2.652,E1 25.0922,E2 35.4122} C_DIS
LIN {X 35.5043,Y 53.8644,Z 75,A 50.8738,B 24.8679,C -2.6528,E1 25.0868,E2 33.1066} C_DIS
LIN {X 33.1466,Y 55.3477,Z 75,A 53.4022,B 24.8674,C -2.6577,E1 25.0808,E2 30.5745} C_DIS
LIN {X 30.8998,Y 56.6318,Z 75,A 55.598,B 24.8673,C -2.6584,E1 25.0755,E2 28.3834} C_DIS
LIN {X 28.6983,Y 57.7784,Z 75,A 58.1199,B 24.8663,C -2.6688,E1 25.0691,E2 25.8438} C_DIS
LIN {X 25.5076,Y 59.2569,Z 75,A 60.9845,B 24.8665,C -2.6661,E1 25.0619,E2 22.9927} C_DIS
LIN {X 21.5507,Y 60.8074,Z 75,A 64.7227,B 24.8663,C -2.6688,E1 25.0521,E2 19.2562} C_DIS
LIN {X 19.0537,Y 61.6351,Z 75,A 67.0575,B 24.8661,C -2.6706,E1 25.0459,E2 16.9215} C_DIS
LIN {X 16.5494,Y 62.3548,Z 75,A 69.3984,B 24.8659,C -2.6727,E1 25.0396,E2 14.5794} C_DIS
LIN {X 14.5865,Y 62.8424,Z 75,A 71.2824,B 24.8656,C -2.6757,E1 25.0345,E2 12.6908} C_DIS
LIN {X 11.8511,Y 63.4161,Z 75,A 73.7267,B 24.8656,C -2.6758,E1 25.0278,E2 10.2491} C_DIS
LIN {X 8.9946,Y 63.883,Z 75,A 76.2482,B 24.8656,C -2.6755,E1 25.0208,E2 7.7309} C_DIS
LIN {X 5.9793,Y 64.2353,Z 75,A 78.9032,B 24.8656,C -2.6749,E1 25.0135,E2 5.079} C_DIS
LIN {X 3.7836,Y 64.4024,Z 75,A 81.422,B 24.8643,C -2.6877,E1 25.0064,E2 2.5309} C_DIS
LIN {X -0.3259,Y 64.5122,Z 75,A 84.6002,B 24.8655,C -2.6764,E1 24.9976,E2 -0.6203} C_DIS
LIN {X -2.7617,Y 64.4539,Z 75,A 86.5545,B 24.866,C -2.6711,E1 24.9921,E2 -2.5622} C_DIS
LIN {X -6.5069,Y 64.1844,Z 75,A 90.3783,B 24.8651,C -2.6804,E1 24.9814,E2 -6.4099} C_DIS
LIN {X -10.1918,Y 63.7038,Z 75,A 93.3668,B 24.866,C -2.6714,E1 24.9732,E2 -9.3794} C_DIS
LIN {X -12.9029,Y 63.2096,Z 75,A 95.7532,B 24.8663,C -2.6681,E1 24.9667,E2 -11.7607} C_DIS
LIN {X -15.8803,Y 62.5282,Z 75,A 98.4888,B 24.8665,C -2.6661,E1 24.9593,E2 -14.4952} C_DIS
LIN {X -18.6243,Y 61.7669,Z 75,A 101.1729,B 24.8665,C -2.6668,E1 24.9521,E2 -17.1852} C_DIS
LIN {X -21.5518,Y 60.807,Z 75,A 104.1939,B 24.8662,C -2.6695,E1 24.9441,E2 -20.2186} C_DIS
LIN {X -25.0391,Y 59.4556,Z 75,A 107.2347,B 24.8672,C -2.659,E1 24.9362,E2 -23.2411} C_DIS
LIN {X -27.9036,Y 58.1663,Z 75,A 109.9834,B 24.8677,C -2.6539,E1 24.9293,E2 -25.9845} C_DIS
LIN {X -32.5069,Y 55.7258,Z 75,A 114.3285,B 24.8691,C -2.6403,E1 24.9187,E2 -30.3094} C_DIS
LIN {X -34.6081,Y 54.4453,Z 75,A 116.7787,B 24.869,C -2.6417,E1 24.9128,E2 -32.7708} C_DIS
LIN {X -37.7326,Y 52.3286,Z 75,A 120.2563,B 24.8694,C -2.6377,E1 24.9049,E2 -36.2506} C_DIS
LIN {X -40.3005,Y 50.378,Z 75,A 123.7775,B 24.8686,C -2.6452,E1 24.8971,E2 -39.8027} C_DIS
LIN {X -43.8646,Y 47.3069,Z 75,A 127.1693,B 24.8711,C -2.6197,E1 24.8901,E2 -43.1472} C_DIS
LIN {X -46.3191,Y 44.9055,Z 75,A 130.1588,B 24.872,C -2.6113,E1 24.8842,E2 -46.1291} C_DIS
LIN {X -49.8897,Y 40.9032,Z 75,A 135.1557,B 24.8727,C -2.6039,E1 24.875,E2 -51.131} C_DIS
LIN {X -52.1911,Y 37.9219,Z 75,A 138.562,B 24.8734,C -2.5963,E1 24.8693,E2 -54.5355} C_DIS
LIN {X -53.9911,Y 35.3121,Z 75,A 141.0736,B 24.8748,C -2.5826,E1 24.8654,E2 -57.0269} C_DIS
LIN {X -55.663,Y 32.6132,Z 75,A 144.3192,B 24.8748,C -2.5831,E1 24.8607,E2 -60.2903} C_DIS
LIN {X -57.7299,Y 28.7961,Z 75,A 147.9507,B 24.8762,C -2.5675,E1 24.856,E2 -63.9039} C_DIS
LIN {X -58.951,Y 26.2071,Z 75,A 150.6334,B 24.8767,C -2.5628,E1 24.8529,E2 -66.5899} C_DIS
LIN {X -59.9565,Y 23.8161,Z 75,A 152.8502,B 24.8775,C -2.5542,E1 24.8505,E2 -68.7985} C_DIS
LIN {X -60.9238,Y 21.219,Z 75,A 155.4068,B 24.8781,C -2.5485,E1 24.8481,E2 -71.3562} C_DIS
LIN {X -61.8126,Y 18.47,Z 75,A 158.2924,B 24.8782,C -2.5469,E1 24.8457,E2 -74.2544} C_DIS
LIN {X -62.7531,Y 14.9695,Z 75,A 160.9494,B 24.8802,C -2.5259,E1 24.8439,E2 -76.8768} C_DIS
LIN {X -63.2324,Y 12.7918,Z 75,A 163.1379,B 24.8804,C -2.5237,E1 24.8427,E2 -79.0729} C_DIS
LIN {X -63.7102,Y 10.1503,Z 75,A 165.5683,B 24.8811,C -2.5171,E1 24.8415,E2 -81.502} C_DIS
LIN {X -64.0624,Y 7.6126,Z 75,A 167.7581,B 24.8819,C -2.5083,E1 24.8407,E2 -83.6838} C_DIS
LIN {X -64.3002,Y 5.237,Z 75,A 170.0392,B 24.8822,C -2.5047,E1 24.8402,E2 -85.9699} C_DIS
LIN {X -64.4645,Y 2.515,Z 75,A 172.5956,B 24.8827,C -2.4996,E1 24.8398,E2 -88.5296} C_DIS
LIN {X -64.512,Y -0.4591,Z 75,A 175.0727,B 24.8838,C -2.4881,E1 24.8398,E2 -90.994} C_DIS
LIN {X -64.4293,Y -3.296,Z 75,A 177.6321,B 24.8845,C -2.4809,E1 24.8401,E2 -93.5517} C_DIS
LIN {X -64.1877,Y -6.4748,Z 75,A -179.5344,B 24.8853,C -2.4721,E1 24.8408,E2 -96.381} C_DIS
LIN {X -63.9109,Y -8.7977,Z 75,A -177.2887,B 24.8856,C -2.4689,E1 24.8416,E2 -98.6327} C_DIS
LIN {X -63.4067,Y -11.9003,Z 75,A -174.5314,B 24.8865,C -2.4596,E1 24.8429,E2 -101.3841} C_DIS
LIN {X -62.7763,Y -14.8726,Z 75,A -171.9166,B 24.8874,C -2.4498,E1 24.8445,E2 -103.9908} C_DIS
LIN {X -62.1117,Y -17.4382,Z 75,A -169.61,B 24.8881,C -2.4418,E1 24.8462,E2 -106.2917} C_DIS
LIN {X -61.4517,Y -19.6384,Z 75,A -167.1674,B 24.8879,C -2.4437,E1 24.8482,E2 -108.7529} C_DIS
LIN {X -59.3768,Y -25.2262,Z 75,A -162.196,B 24.8899,C -2.4221,E1 24.8532,E2 -113.7006} C_DIS
LIN {X -58.2258,Y -27.7799,Z 75,A -159.7001,B 24.8905,C -2.4153,E1 24.8561,E2 -116.194} C_DIS
LIN {X -57.1896,Y -29.8553,Z 75,A -157.8409,B 24.8914,C -2.4057,E1 24.8585,E2 -118.0401} C_DIS
LIN {X -56.2222,Y -31.6392,Z 75,A -155.6216,B 24.8911,C -2.4093,E1 24.8615,E2 -120.2797} C_DIS
LIN {X -54.8497,Y -33.9633,Z 75,A -153.3287,B 24.8918,C -2.401,E1 24.8648,E2 -122.5644} C_DIS
Enddeposition()
END
